LIN {X 0,Y 525.417,Z 230.64,A -85,B 0,C 180,E1 -4783.488,E2 -4783.488} C_VEL
LIN {X 0,Y 525.578,Z 217.368,A -85,B 0,C 180,E1 -4783.73,E2 -4783.73} C_VEL
LIN {X 0,Y 525.769,Z 127.353,A -85,B 0,C 180,E1 -4784.968,E2 -4784.968} C_VEL
LIN {X 0,Y 524.225,Z 116.388,A -85,B 0,C 180,E1 -4785.187,E2 -4785.187} C_VEL
LIN {X 0,Y 524.577,Z 97.639,A -85,B 0,C 180,E1 -4787.969,E2 -4787.969} C_VEL
LIN {X 0,Y 525.034,Z 77.543,A -85,B 0,C 180,E1 -4790.981,E2 -4790.981} C_VEL
LIN {X 0,Y 525.375,Z 61.269,A -85,B 0,C 180,E1 -4793.451,E2 -4793.451} C_VEL
LIN {X 0,Y 525.033,Z 57.51,A -85,B 0,C 180,E1 -4794.042,E2 -4794.042} C_VEL
LIN {X 0,Y 523.985,Z 52.216,A -85,B 0,C 180,E1 -4794.939,E2 -4794.939} C_VEL
LIN {X 0,Y 523.971,Z 52.218,A -85,B 0,C 180,E1 -4797.999,E2 -4797.999} C_VEL
LIN {X 0,Y 523.946,Z 52.215,A -85,B 0,C 180,E1 -4800.854,E2 -4800.854} C_VEL
LIN {X 0,Y 523.96,Z 52.22,A -85,B 0,C 180,E1 -4803.734,E2 -4803.734} C_VEL
LIN {X 0,Y 523.904,Z 52.222,A -85,B 0,C 180,E1 -4806.401,E2 -4806.401} C_VEL
LIN {X 0,Y 523.923,Z 52.219,A -85,B 0,C 180,E1 -4809.084,E2 -4809.084} C_VEL
LIN {X 0,Y 523.951,Z 52.217,A -85,B 0,C 180,E1 -4812.119,E2 -4812.119} C_VEL
LIN {X 0,Y 523.942,Z 52.222,A -85,B 0,C 180,E1 -4815.31,E2 -4815.31} C_VEL
LIN {X 0,Y 523.955,Z 52.215,A -85,B 0,C 180,E1 -4818.69,E2 -4818.69} C_VEL
LIN {X 0,Y 523.916,Z 52.224,A -85,B 0,C 180,E1 -4821.081,E2 -4821.081} C_VEL
LIN {X 0,Y 523.902,Z 52.222,A -85,B 0,C 180,E1 -4823.825,E2 -4823.825} C_VEL
LIN {X 0,Y 523.941,Z 52.218,A -85,B 0,C 180,E1 -4826.636,E2 -4826.636} C_VEL
LIN {X 0,Y 523.956,Z 52.218,A -85,B 0,C 180,E1 -4829.356,E2 -4829.356} C_VEL
LIN {X 0,Y 523.976,Z 52.212,A -85,B 0,C 180,E1 -4832.281,E2 -4832.281} C_VEL
LIN {X 0,Y 523.947,Z 52.219,A -85,B 0,C 180,E1 -4834.581,E2 -4834.581} C_VEL
LIN {X 0,Y 523.918,Z 52.218,A -85,B 0,C 180,E1 -4837.757,E2 -4837.757} C_VEL
LIN {X 0,Y 523.974,Z 52.216,A -85,B 0,C 180,E1 -4840.408,E2 -4840.408} C_VEL
LIN {X 0,Y 523.953,Z 52.22,A -85,B 0,C 180,E1 -4842.837,E2 -4842.837} C_VEL
LIN {X 0,Y 523.975,Z 52.212,A -85,B 0,C 180,E1 -4845.236,E2 -4845.236} C_VEL
LIN {X 0,Y 524.013,Z 52.215,A -85,B 0,C 180,E1 -4848.394,E2 -4848.394} C_VEL
LIN {X 0,Y 523.999,Z 52.209,A -85,B 0,C 180,E1 -4851.516,E2 -4851.516} C_VEL
LIN {X 0,Y 524.078,Z 52.202,A -85,B 0,C 180,E1 -4854.614,E2 -4854.614} C_VEL
LIN {X 0,Y 524.111,Z 52.197,A -85,B 0,C 180,E1 -4857.695,E2 -4857.695} C_VEL
LIN {X 0,Y 524.119,Z 52.194,A -85,B 0,C 180,E1 -4860.768,E2 -4860.768} C_VEL
LIN {X 0,Y 524.042,Z 52.203,A -85,B 0,C 180,E1 -4863.075,E2 -4863.075} C_VEL
LIN {X 0,Y 524.027,Z 52.21,A -85,B 0,C 180,E1 -4866.159,E2 -4866.159} C_VEL
LIN {X 0,Y 523.986,Z 52.212,A -85,B 0,C 180,E1 -4869.262,E2 -4869.262} C_VEL
LIN {X 0,Y 524,Z 52.217,A -85,B 0,C 180,E1 -4871.738,E2 -4871.738} C_VEL
LIN {X 0,Y 523.992,Z 52.211,A -85,B 0,C 180,E1 -4875.052,E2 -4875.052} C_VEL
LIN {X 0,Y 523.945,Z 52.218,A -85,B 0,C 180,E1 -4877.97,E2 -4877.97} C_VEL
LIN {X 0,Y 523.958,Z 52.213,A -85,B 0,C 180,E1 -4880.411,E2 -4880.411} C_VEL
LIN {X 0,Y 523.908,Z 52.222,A -85,B 0,C 180,E1 -4882.894,E2 -4882.894} C_VEL
LIN {X 0,Y 523.914,Z 52.226,A -85,B 0,C 180,E1 -4885.421,E2 -4885.421} C_VEL
LIN {X 0,Y 523.958,Z 52.214,A -85,B 0,C 180,E1 -4888,E2 -4888} C_VEL
LIN {X 0,Y 523.939,Z 52.221,A -85,B 0,C 180,E1 -4890.854,E2 -4890.854} C_VEL
LIN {X 0,Y 523.93,Z 52.218,A -85,B 0,C 180,E1 -4893.73,E2 -4893.73} C_VEL
LIN {X 0,Y 523.904,Z 52.222,A -85,B 0,C 180,E1 -4896.402,E2 -4896.402} C_VEL
LIN {X 0,Y 523.914,Z 52.225,A -85,B 0,C 180,E1 -4899.086,E2 -4899.086} C_VEL
LIN {X 0,Y 523.91,Z 52.221,A -85,B 0,C 180,E1 -4902.124,E2 -4902.124} C_VEL
LIN {X 0,Y 523.942,Z 52.217,A -85,B 0,C 180,E1 -4905.311,E2 -4905.311} C_VEL
LIN {X 0,Y 523.902,Z 52.225,A -85,B 0,C 180,E1 -4906.885,E2 -4906.885} C_VEL
LIN {X 0,Y 523.23,Z 52.307,A -85,B 0,C 180,E1 -4907.527,E2 -4907.527} C_VEL
LIN {X 0,Y 520.367,Z 52.67,A -85,B 0,C 180,E1 -4908.568,E2 -4908.568} C_VEL
LIN {X 0,Y 517.961,Z 52.965,A -85,B 0,C 180,E1 -4909.407,E2 -4909.407} C_VEL
LIN {X 0,Y 516.947,Z 53.09,A -85,B 0,C 180,E1 -4910.055,E2 -4910.055} C_VEL
LIN {X 0,Y 516.875,Z 53.101,A -85,B 0,C 180,E1 -4910.274,E2 -4910.274} C_VEL
LIN {X 0,Y 516.85,Z 53.099,A -85,B 0,C 180,E1 -4913.348,E2 -4913.348} C_VEL
LIN {X 0,Y 516.902,Z 53.098,A -85,B 0,C 180,E1 -4916.12,E2 -4916.12} C_VEL
LIN {X 0,Y 516.895,Z 53.094,A -85,B 0,C 180,E1 -4918.936,E2 -4918.936} C_VEL
LIN {X 0,Y 516.863,Z 53.099,A -85,B 0,C 180,E1 -4921.582,E2 -4921.582} C_VEL
LIN {X 0,Y 516.872,Z 53.103,A -85,B 0,C 180,E1 -4924.208,E2 -4924.208} C_VEL
LIN {X 0,Y 516.862,Z 53.098,A -85,B 0,C 180,E1 -4926.776,E2 -4926.776} C_VEL
LIN {X 0,Y 516.942,Z 53.094,A -85,B 0,C 180,E1 -4929.733,E2 -4929.733} C_VEL
LIN {X 0,Y 516.889,Z 53.095,A -85,B 0,C 180,E1 -4932.595,E2 -4932.595} C_VEL
LIN {X 0,Y 516.944,Z 53.091,A -85,B 0,C 180,E1 -4935.03,E2 -4935.03} C_VEL
LIN {X 0,Y 516.966,Z 53.271,A -85,B 0,C 180,E1 -4937.756,E2 -4937.756} C_VEL
LIN {X 0,Y 517.485,Z 57.551,A -85,B 0,C 180,E1 -4938.643,E2 -4938.643} C_VEL
LIN {X 0,Y 517.416,Z 69.345,A -85,B 0,C 180,E1 -4941.014,E2 -4941.014} C_VEL
LIN {X 0,Y 517.278,Z 72.801,A -85,B 0,C 180,E1 -4941.696,E2 -4941.696} C_VEL
LIN {X 0,Y 519.153,Z 83.02,A -85,B 0,C 180,E1 -4941.901,E2 -4941.901} C_VEL
LIN {X 0,Y 518.614,Z 179.674,A -85,B 0,C 180,E1 -4943.264,E2 -4943.264} C_VEL
LIN {X 0,Y 518.437,Z 193.363,A -85,B 0,C 180,E1 -4943.628,E2 -4943.628} C_VEL
LIN {X 0,Y 518.283,Z 205.634,A -85,B 0,C 180,E1 -4944.114,E2 -4944.114} C_VEL
LIN {X 0,Y 518.082,Z 217.393,A -85,B 0,C 180,E1 -4944.746,E2 -4944.746} C_VEL
LIN {X 0,Y 517.745,Z 228.688,A -85,B 0,C 180,E1 -4945.524,E2 -4945.524} C_VEL
LIN {X 0,Y 517.419,Z 238.884,A -85,B 0,C 180,E1 -4946.399,E2 -4946.399} C_VEL
LIN {X 0,Y 517.184,Z 247.231,A -85,B 0,C 180,E1 -4947.274,E2 -4947.274} C_VEL
LIN {X 0,Y 516.859,Z 256.313,A -85,B 0,C 180,E1 -4948.442,E2 -4948.442} C_VEL
LIN {X 0,Y 516.712,Z 263.613,A -85,B 0,C 180,E1 -4949.611,E2 -4949.611} C_VEL
LIN {X 0,Y 516.473,Z 269.502,A -85,B 0,C 180,E1 -4950.78,E2 -4950.78} C_VEL
LIN {X 0,Y 516.401,Z 274.157,A -85,B 0,C 180,E1 -4951.95,E2 -4951.95} C_VEL
LIN {X 0,Y 516.389,Z 277.725,A -85,B 0,C 180,E1 -4953.121,E2 -4953.121} C_VEL
LIN {X 0,Y 516.332,Z 279.576,A -85,B 0,C 180,E1 -4953.903,E2 -4953.903} C_VEL
LIN {X 0,Y 516.247,Z 280.97,A -85,B 0,C 180,E1 -4954.685,E2 -4954.685} C_VEL
LIN {X 0,Y 516.312,Z 281.956,A -85,B 0,C 180,E1 -4955.468,E2 -4955.468} C_VEL
LIN {X 0,Y 516.374,Z 282.679,A -85,B 0,C 180,E1 -4956.506,E2 -4956.506} C_VEL
LIN {X 0,Y 516.279,Z 282.577,A -85,B 0,C 180,E1 -4957.824,E2 -4957.824} C_VEL
LIN {X 0,Y 516.23,Z 280.982,A -85,B 0,C 180,E1 -4959.403,E2 -4959.403} C_VEL
LIN {X 0,Y 516.294,Z 279.577,A -85,B 0,C 180,E1 -4960.193,E2 -4960.193} C_VEL
LIN {X 0,Y 516.366,Z 276.299,A -85,B 0,C 180,E1 -4961.488,E2 -4961.488} C_VEL
LIN {X 0,Y 516.474,Z 272.599,A -85,B 0,C 180,E1 -4962.576,E2 -4962.576} C_VEL
LIN {X 0,Y 516.644,Z 266.35,A -85,B 0,C 180,E1 -4963.973,E2 -4963.973} C_VEL
LIN {X 0,Y 516.797,Z 260.069,A -85,B 0,C 180,E1 -4965.083,E2 -4965.083} C_VEL
LIN {X 0,Y 517.008,Z 252.455,A -85,B 0,C 180,E1 -4966.181,E2 -4966.181} C_VEL
LIN {X 0,Y 517.251,Z 243.92,A -85,B 0,C 180,E1 -4967.189,E2 -4967.189} C_VEL
LIN {X 0,Y 517.561,Z 233.283,A -85,B 0,C 180,E1 -4968.199,E2 -4968.199} C_VEL
LIN {X 0,Y 517.868,Z 222.67,A -85,B 0,C 180,E1 -4969.009,E2 -4969.009} C_VEL
LIN {X 0,Y 518.182,Z 210.921,A -85,B 0,C 180,E1 -4969.717,E2 -4969.717} C_VEL
LIN {X 0,Y 518.418,Z 198.575,A -85,B 0,C 180,E1 -4970.276,E2 -4970.276} C_VEL
LIN {X 0,Y 518.614,Z 186.111,A -85,B 0,C 180,E1 -4970.678,E2 -4970.678} C_VEL
LIN {X 0,Y 518.725,Z 174.043,A -85,B 0,C 180,E1 -4970.924,E2 -4970.924} C_VEL
LIN {X 0,Y 519.058,Z 81.453,A -85,B 0,C 180,E1 -4972.218,E2 -4972.218} C_VEL
LIN {X 0,Y 517.329,Z 72.818,A -85,B 0,C 180,E1 -4972.41,E2 -4972.41} C_VEL
LIN {X 0,Y 517.6,Z 58.332,A -85,B 0,C 180,E1 -4975.323,E2 -4975.323} C_VEL
LIN {X 0,Y 516.886,Z 53.103,A -85,B 0,C 180,E1 -4976.462,E2 -4976.462} C_VEL
LIN {X 0,Y 516.889,Z 53.098,A -85,B 0,C 180,E1 -4979.518,E2 -4979.518} C_VEL
LIN {X 0,Y 516.868,Z 53.104,A -85,B 0,C 180,E1 -4982.538,E2 -4982.538} C_VEL
LIN {X 0,Y 516.831,Z 53.103,A -85,B 0,C 180,E1 -4985.323,E2 -4985.323} C_VEL
LIN {X 0,Y 516.862,Z 53.1,A -85,B 0,C 180,E1 -4988.718,E2 -4988.718} C_VEL
LIN {X 0,Y 516.834,Z 53.109,A -85,B 0,C 180,E1 -4991.783,E2 -4991.783} C_VEL
LIN {X 0,Y 516.9,Z 53.089,A -85,B 0,C 180,E1 -4995.007,E2 -4995.007} C_VEL
LIN {X 0,Y 516.832,Z 53.101,A -85,B 0,C 180,E1 -4998.409,E2 -4998.409} C_VEL
LIN {X 0,Y 516.849,Z 53.104,A -85,B 0,C 180,E1 -5001.281,E2 -5001.281} C_VEL
LIN {X 0,Y 516.83,Z 53.101,A -85,B 0,C 180,E1 -5004.677,E2 -5004.677} C_VEL
LIN {X 0,Y 516.867,Z 53.102,A -85,B 0,C 180,E1 -5007.462,E2 -5007.462} C_VEL
LIN {X 0,Y 516.848,Z 53.1,A -85,B 0,C 180,E1 -5010.489,E2 -5010.489} C_VEL
LIN {X 0,Y 516.829,Z 53.108,A -85,B 0,C 180,E1 -5013.337,E2 -5013.337} C_VEL
LIN {X 0,Y 516.871,Z 53.096,A -85,B 0,C 180,E1 -5015.926,E2 -5015.926} C_VEL
LIN {X 0,Y 516.886,Z 53.095,A -85,B 0,C 180,E1 -5018.462,E2 -5018.462} C_VEL
LIN {X 0,Y 516.888,Z 53.1,A -85,B 0,C 180,E1 -5020.954,E2 -5020.954} C_VEL
LIN {X 0,Y 516.882,Z 53.096,A -85,B 0,C 180,E1 -5023.409,E2 -5023.409} C_VEL
LIN {X 0,Y 516.872,Z 53.097,A -85,B 0,C 180,E1 -5025.833,E2 -5025.833} C_VEL
LIN {X 0,Y 516.946,Z 53.089,A -85,B 0,C 180,E1 -5029.028,E2 -5029.028} C_VEL
LIN {X 0,Y 516.93,Z 53.094,A -85,B 0,C 180,E1 -5032.186,E2 -5032.186} C_VEL
LIN {X 0,Y 516.983,Z 53.088,A -85,B 0,C 180,E1 -5034.539,E2 -5034.539} C_VEL
LIN {X 0,Y 517.077,Z 53.073,A -85,B 0,C 180,E1 -5037.663,E2 -5037.663} C_VEL
LIN {X 0,Y 517.092,Z 53.069,A -85,B 0,C 180,E1 -5040.779,E2 -5040.779} C_VEL
LIN {X 0,Y 516.949,Z 53.087,A -85,B 0,C 180,E1 -5043.117,E2 -5043.117} C_VEL
LIN {X 0,Y 516.976,Z 53.086,A -85,B 0,C 180,E1 -5046.243,E2 -5046.243} C_VEL
LIN {X 0,Y 516.941,Z 53.091,A -85,B 0,C 180,E1 -5049.389,E2 -5049.389} C_VEL
LIN {X 0,Y 516.956,Z 53.09,A -85,B 0,C 180,E1 -5051.807,E2 -5051.807} C_VEL
LIN {X 0,Y 516.942,Z 53.09,A -85,B 0,C 180,E1 -5055.144,E2 -5055.144} C_VEL
LIN {X 0,Y 516.881,Z 53.095,A -85,B 0,C 180,E1 -5058.224,E2 -5058.224} C_VEL
LIN {X 0,Y 516.908,Z 53.092,A -85,B 0,C 180,E1 -5060.702,E2 -5060.702} C_VEL
LIN {X 0,Y 516.888,Z 53.095,A -85,B 0,C 180,E1 -5064.073,E2 -5064.073} C_VEL
LIN {X 0,Y 516.907,Z 53.093,A -85,B 0,C 180,E1 -5066.659,E2 -5066.659} C_VEL
LIN {X 0,Y 516.91,Z 53.095,A -85,B 0,C 180,E1 -5069.523,E2 -5069.523} C_VEL
LIN {X 0,Y 516.899,Z 53.095,A -85,B 0,C 180,E1 -5072.543,E2 -5072.543} C_VEL
LIN {X 0,Y 516.871,Z 53.094,A -85,B 0,C 180,E1 -5075.33,E2 -5075.33} C_VEL
LIN {X 0,Y 516.882,Z 53.093,A -85,B 0,C 180,E1 -5077.943,E2 -5077.943} C_VEL
LIN {X 0,Y 516.886,Z 53.102,A -85,B 0,C 180,E1 -5080.742,E2 -5080.742} C_VEL
LIN {X 0,Y 516.885,Z 53.102,A -85,B 0,C 180,E1 -5082.831,E2 -5082.831} C_VEL
LIN {X 0,Y 516.898,Z 53.096,A -85,B 0,C 180,E1 -5085.007,E2 -5085.007} C_VEL
LIN {X 0,Y 516.916,Z 53.097,A -85,B 0,C 180,E1 -5088.399,E2 -5088.399} C_VEL
LIN {X 0,Y 516.884,Z 53.095,A -85,B 0,C 180,E1 -5091.284,E2 -5091.284} C_VEL
LIN {X 0,Y 516.874,Z 53.102,A -85,B 0,C 180,E1 -5094.22,E2 -5094.22} C_VEL
LIN {X 0,Y 516.898,Z 53.097,A -85,B 0,C 180,E1 -5097.053,E2 -5097.053} C_VEL
LIN {X 0,Y 516.895,Z 53.102,A -85,B 0,C 180,E1 -5099.796,E2 -5099.796} C_VEL
LIN {X 0,Y 516.929,Z 53.094,A -85,B 0,C 180,E1 -5102.467,E2 -5102.467} C_VEL
LIN {X 0,Y 516.939,Z 53.134,A -85,B 0,C 180,E1 -5104.858,E2 -5104.858} C_VEL
LIN {X 0,Y 518.443,Z 61.217,A -85,B 0,C 180,E1 -5106.216,E2 -5106.216} C_VEL
LIN {X 0,Y 518.131,Z 74.628,A -85,B 0,C 180,E1 -5108.307,E2 -5108.307} C_VEL
LIN {X 0,Y 517.731,Z 90.731,A -85,B 0,C 180,E1 -5110.78,E2 -5110.78} C_VEL
LIN {X 0,Y 517.337,Z 109.522,A -85,B 0,C 180,E1 -5113.627,E2 -5113.627} C_VEL
LIN {X 0,Y 517.18,Z 116.074,A -85,B 0,C 180,E1 -5114.61,E2 -5114.61} C_VEL
LIN {X 0,Y 519.009,Z 129.152,A -85,B 0,C 180,E1 -5114.863,E2 -5114.863} C_VEL
LIN {X 0,Y 518.575,Z 224.633,A -85,B 0,C 180,E1 -5116.205,E2 -5116.205} C_VEL
LIN {X 0,Y 518.337,Z 237.966,A -85,B 0,C 180,E1 -5116.549,E2 -5116.549} C_VEL
LIN {X 0,Y 518.029,Z 251.299,A -85,B 0,C 180,E1 -5117.064,E2 -5117.064} C_VEL
LIN {X 0,Y 517.755,Z 263.311,A -85,B 0,C 180,E1 -5117.706,E2 -5117.706} C_VEL
LIN {X 0,Y 517.445,Z 274.128,A -85,B 0,C 180,E1 -5118.443,E2 -5118.443} C_VEL
LIN {X 0,Y 517.173,Z 284.608,A -85,B 0,C 180,E1 -5119.33,E2 -5119.33} C_VEL
LIN {X 0,Y 516.878,Z 293.178,A -85,B 0,C 180,E1 -5120.214,E2 -5120.214} C_VEL
LIN {X 0,Y 516.672,Z 301.089,A -85,B 0,C 180,E1 -5121.197,E2 -5121.197} C_VEL
LIN {X 0,Y 516.511,Z 308.82,A -85,B 0,C 180,E1 -5122.376,E2 -5122.376} C_VEL
LIN {X 0,Y 516.353,Z 315.946,A -85,B 0,C 180,E1 -5123.749,E2 -5123.749} C_VEL
LIN {X 0,Y 516.311,Z 320.69,A -85,B 0,C 180,E1 -5124.924,E2 -5124.924} C_VEL
LIN {X 0,Y 516.351,Z 324.319,A -85,B 0,C 180,E1 -5126.098,E2 -5126.098} C_VEL
LIN {X 0,Y 516.303,Z 326.188,A -85,B 0,C 180,E1 -5126.879,E2 -5126.879} C_VEL
LIN {X 0,Y 516.264,Z 327.59,A -85,B 0,C 180,E1 -5127.659,E2 -5127.659} C_VEL
LIN {X 0,Y 516.177,Z 329.2,A -85,B 0,C 180,E1 -5129.22,E2 -5129.22} C_VEL
LIN {X 0,Y 516.179,Z 329.419,A -85,B 0,C 180,E1 -5130,E2 -5130} C_VEL
LIN {X 0,Y 516.196,Z 328.597,A -85,B 0,C 180,E1 -5131.56,E2 -5131.56} C_VEL
LIN {X 0,Y 516.264,Z 327.603,A -85,B 0,C 180,E1 -5132.34,E2 -5132.34} C_VEL
LIN {X 0,Y 516.303,Z 326.205,A -85,B 0,C 180,E1 -5133.121,E2 -5133.121} C_VEL
LIN {X 0,Y 516.309,Z 323.26,A -85,B 0,C 180,E1 -5134.293,E2 -5134.293} C_VEL
LIN {X 0,Y 516.364,Z 319.275,A -85,B 0,C 180,E1 -5135.467,E2 -5135.467} C_VEL
LIN {X 0,Y 516.414,Z 313.144,A -85,B 0,C 180,E1 -5136.839,E2 -5136.839} C_VEL
LIN {X 0,Y 516.561,Z 306.446,A -85,B 0,C 180,E1 -5138.016,E2 -5138.016} C_VEL
LIN {X 0,Y 516.741,Z 298.137,A -85,B 0,C 180,E1 -5139.195,E2 -5139.195} C_VEL
LIN {X 0,Y 516.947,Z 289.622,A -85,B 0,C 180,E1 -5140.18,E2 -5140.18} C_VEL
LIN {X 0,Y 517.29,Z 279.107,A -85,B 0,C 180,E1 -5141.163,E2 -5141.163} C_VEL
LIN {X 0,Y 517.607,Z 267.374,A -85,B 0,C 180,E1 -5142.043,E2 -5142.043} C_VEL
LIN {X 0,Y 517.946,Z 255.379,A -85,B 0,C 180,E1 -5142.738,E2 -5142.738} C_VEL
LIN {X 0,Y 518.209,Z 243.005,A -85,B 0,C 180,E1 -5143.28,E2 -5143.28} C_VEL
LIN {X 0,Y 518.53,Z 230.312,A -85,B 0,C 180,E1 -5143.671,E2 -5143.671} C_VEL
LIN {X 0,Y 518.677,Z 217.028,A -85,B 0,C 180,E1 -5143.916,E2 -5143.916} C_VEL
LIN {X 0,Y 518.96,Z 128.491,A -85,B 0,C 180,E1 -5145.149,E2 -5145.149} C_VEL
LIN {X 0,Y 517.219,Z 116.148,A -85,B 0,C 180,E1 -5145.387,E2 -5145.387} C_VEL
LIN {X 0,Y 517.662,Z 96.105,A -85,B 0,C 180,E1 -5148.4,E2 -5148.4} C_VEL
LIN {X 0,Y 518.122,Z 75.816,A -85,B 0,C 180,E1 -5151.484,E2 -5151.484} C_VEL
LIN {X 0,Y 518.441,Z 62.24,A -85,B 0,C 180,E1 -5153.572,E2 -5153.572} C_VEL
LIN {X 0,Y 517.434,Z 55.557,A -85,B 0,C 180,E1 -5154.656,E2 -5154.656} C_VEL
LIN {X 0,Y 516.948,Z 53.092,A -85,B 0,C 180,E1 -5155.087,E2 -5155.087} C_VEL
LIN {X 0,Y 516.928,Z 53.094,A -85,B 0,C 180,E1 -5157.905,E2 -5157.905} C_VEL
LIN {X 0,Y 516.893,Z 53.1,A -85,B 0,C 180,E1 -5160.203,E2 -5160.203} C_VEL
LIN {X 0,Y 516.896,Z 53.093,A -85,B 0,C 180,E1 -5162.947,E2 -5162.947} C_VEL
LIN {X 0,Y 516.872,Z 53.105,A -85,B 0,C 180,E1 -5165.78,E2 -5165.78} C_VEL
LIN {X 0,Y 516.883,Z 53.095,A -85,B 0,C 180,E1 -5168.715,E2 -5168.715} C_VEL
LIN {X 0,Y 516.912,Z 53.098,A -85,B 0,C 180,E1 -5171.775,E2 -5171.775} C_VEL
LIN {X 0,Y 516.895,Z 53.096,A -85,B 0,C 180,E1 -5175.007,E2 -5175.007} C_VEL
LIN {X 0,Y 516.913,Z 53.091,A -85,B 0,C 180,E1 -5178.399,E2 -5178.399} C_VEL
LIN {X 0,Y 516.879,Z 53.104,A -85,B 0,C 180,E1 -5181.284,E2 -5181.284} C_VEL
LIN {X 0,Y 516.873,Z 53.096,A -85,B 0,C 180,E1 -5184.22,E2 -5184.22} C_VEL
LIN {X 0,Y 516.895,Z 53.101,A -85,B 0,C 180,E1 -5187.053,E2 -5187.053} C_VEL
LIN {X 0,Y 516.891,Z 53.094,A -85,B 0,C 180,E1 -5189.796,E2 -5189.796} C_VEL
LIN {X 0,Y 516.926,Z 53.092,A -85,B 0,C 180,E1 -5192.467,E2 -5192.467} C_VEL
LIN {X 0,Y 516.903,Z 53.098,A -85,B 0,C 180,E1 -5195.072,E2 -5195.072} C_VEL
LIN {X 0,Y 516.885,Z 53.099,A -85,B 0,C 180,E1 -5198.462,E2 -5198.462} C_VEL
LIN {X 0,Y 516.9,Z 53.098,A -85,B 0,C 180,E1 -5200.955,E2 -5200.955} C_VEL
LIN {X 0,Y 516.903,Z 53.093,A -85,B 0,C 180,E1 -5203.41,E2 -5203.41} C_VEL
LIN {X 0,Y 516.891,Z 53.095,A -85,B 0,C 180,E1 -5205.834,E2 -5205.834} C_VEL
LIN {X 0,Y 516.95,Z 53.088,A -85,B 0,C 180,E1 -5209.028,E2 -5209.028} C_VEL
LIN {X 0,Y 516.977,Z 53.09,A -85,B 0,C 180,E1 -5212.187,E2 -5212.187} C_VEL
LIN {X 0,Y 517.026,Z 53.082,A -85,B 0,C 180,E1 -5214.54,E2 -5214.54} C_VEL
LIN {X 0,Y 517.082,Z 53.072,A -85,B 0,C 180,E1 -5217.663,E2 -5217.663} C_VEL
LIN {X 0,Y 517.09,Z 53.07,A -85,B 0,C 180,E1 -5220.779,E2 -5220.779} C_VEL
LIN {X 0,Y 516.985,Z 53.082,A -85,B 0,C 180,E1 -5223.117,E2 -5223.117} C_VEL
LIN {X 0,Y 516.989,Z 53.086,A -85,B 0,C 180,E1 -5226.244,E2 -5226.244} C_VEL
LIN {X 0,Y 516.942,Z 53.091,A -85,B 0,C 180,E1 -5229.39,E2 -5229.39} C_VEL
LIN {X 0,Y 516.952,Z 53.094,A -85,B 0,C 180,E1 -5231.807,E2 -5231.807} C_VEL
LIN {X 0,Y 516.943,Z 53.09,A -85,B 0,C 180,E1 -5235.146,E2 -5235.146} C_VEL
LIN {X 0,Y 516.913,Z 53.092,A -85,B 0,C 180,E1 -5238.223,E2 -5238.223} C_VEL
LIN {X 0,Y 516.905,Z 53.093,A -85,B 0,C 180,E1 -5240.702,E2 -5240.702} C_VEL
LIN {X 0,Y 516.886,Z 53.095,A -85,B 0,C 180,E1 -5244.074,E2 -5244.074} C_VEL
LIN {X 0,Y 516.908,Z 53.093,A -85,B 0,C 180,E1 -5246.659,E2 -5246.659} C_VEL
LIN {X 0,Y 516.909,Z 53.095,A -85,B 0,C 180,E1 -5249.524,E2 -5249.524} C_VEL
LIN {X 0,Y 516.895,Z 53.096,A -85,B 0,C 180,E1 -5252.543,E2 -5252.543} C_VEL
LIN {X 0,Y 516.866,Z 53.101,A -85,B 0,C 180,E1 -5255.33,E2 -5255.33} C_VEL
LIN {X 0,Y 516.88,Z 53.095,A -85,B 0,C 180,E1 -5257.943,E2 -5257.943} C_VEL
LIN {X 0,Y 516.854,Z 53.107,A -85,B 0,C 180,E1 -5260.745,E2 -5260.745} C_VEL
LIN {X 0,Y 516.882,Z 53.095,A -85,B 0,C 180,E1 -5263.904,E2 -5263.904} C_VEL
LIN {X 0,Y 516.849,Z 53.099,A -85,B 0,C 180,E1 -5266.887,E2 -5266.887} C_VEL
LIN {X 0,Y 516.882,Z 53.095,A -85,B 0,C 180,E1 -5269.591,E2 -5269.591} C_VEL
LIN {X 0,Y 516.875,Z 53.101,A -85,B 0,C 180,E1 -5270.274,E2 -5270.274} C_VEL
LIN {X 0,Y 516.232,Z 53.187,A -85,B 0,C 180,E1 -5270.925,E2 -5270.925} C_VEL
LIN {X 0,Y 513.378,Z 53.54,A -85,B 0,C 180,E1 -5271.98,E2 -5271.98} C_VEL
LIN {X 0,Y 510.944,Z 53.838,A -85,B 0,C 180,E1 -5272.83,E2 -5272.83} C_VEL
LIN {X 0,Y 509.892,Z 53.966,A -85,B 0,C 180,E1 -5273.487,E2 -5273.487} C_VEL
LIN {X 0,Y 509.804,Z 53.977,A -85,B 0,C 180,E1 -5273.709,E2 -5273.709} C_VEL
LIN {X 0,Y 509.855,Z 53.976,A -85,B 0,C 180,E1 -5276.539,E2 -5276.539} C_VEL
LIN {X 0,Y 509.849,Z 53.971,A -85,B 0,C 180,E1 -5279.335,E2 -5279.335} C_VEL
LIN {X 0,Y 509.847,Z 53.979,A -85,B 0,C 180,E1 -5282.052,E2 -5282.052} C_VEL
LIN {X 0,Y 509.804,Z 53.978,A -85,B 0,C 180,E1 -5284.7,E2 -5284.7} C_VEL
LIN {X 0,Y 509.83,Z 53.976,A -85,B 0,C 180,E1 -5287.459,E2 -5287.459} C_VEL
LIN {X 0,Y 509.919,Z 53.971,A -85,B 0,C 180,E1 -5289.845,E2 -5289.845} C_VEL
LIN {X 0,Y 509.86,Z 53.971,A -85,B 0,C 180,E1 -5293.174,E2 -5293.174} C_VEL
LIN {X 0,Y 509.858,Z 53.979,A -85,B 0,C 180,E1 -5295.634,E2 -5295.634} C_VEL
LIN {X 0,Y 509.908,Z 54.059,A -85,B 0,C 180,E1 -5297.615,E2 -5297.615} C_VEL
LIN {X 0,Y 510.464,Z 58.208,A -85,B 0,C 180,E1 -5298.485,E2 -5298.485} C_VEL
LIN {X 0,Y 510.427,Z 70.066,A -85,B 0,C 180,E1 -5300.89,E2 -5300.89} C_VEL
LIN {X 0,Y 510.297,Z 73.056,A -85,B 0,C 180,E1 -5301.484,E2 -5301.484} C_VEL
LIN {X 0,Y 512.301,Z 83.987,A -85,B 0,C 180,E1 -5301.709,E2 -5301.709} C_VEL
LIN {X 0,Y 511.733,Z 179.747,A -85,B 0,C 180,E1 -5303.074,E2 -5303.074} C_VEL
LIN {X 0,Y 511.565,Z 192.771,A -85,B 0,C 180,E1 -5303.418,E2 -5303.418} C_VEL
LIN {X 0,Y 511.376,Z 205.848,A -85,B 0,C 180,E1 -5303.936,E2 -5303.936} C_VEL
LIN {X 0,Y 511.153,Z 217.649,A -85,B 0,C 180,E1 -5304.576,E2 -5304.576} C_VEL
LIN {X 0,Y 510.799,Z 228.966,A -85,B 0,C 180,E1 -5305.364,E2 -5305.364} C_VEL
LIN {X 0,Y 510.453,Z 239.172,A -85,B 0,C 180,E1 -5306.25,E2 -5306.25} C_VEL
LIN {X 0,Y 510.155,Z 248.374,A -85,B 0,C 180,E1 -5307.237,E2 -5307.237} C_VEL
LIN {X 0,Y 509.814,Z 257.287,A -85,B 0,C 180,E1 -5308.42,E2 -5308.42} C_VEL
LIN {X 0,Y 509.668,Z 264.473,A -85,B 0,C 180,E1 -5309.605,E2 -5309.605} C_VEL
LIN {X 0,Y 509.397,Z 270.263,A -85,B 0,C 180,E1 -5310.791,E2 -5310.791} C_VEL
LIN {X 0,Y 509.336,Z 274.823,A -85,B 0,C 180,E1 -5311.977,E2 -5311.977} C_VEL
LIN {X 0,Y 509.325,Z 278.304,A -85,B 0,C 180,E1 -5313.164,E2 -5313.164} C_VEL
LIN {X 0,Y 509.258,Z 280.083,A -85,B 0,C 180,E1 -5313.957,E2 -5313.957} C_VEL
LIN {X 0,Y 509.162,Z 281.428,A -85,B 0,C 180,E1 -5314.751,E2 -5314.751} C_VEL
LIN {X 0,Y 509.245,Z 282.373,A -85,B 0,C 180,E1 -5315.544,E2 -5315.544} C_VEL
LIN {X 0,Y 509.291,Z 282.998,A -85,B 0,C 180,E1 -5316.497,E2 -5316.497} C_VEL
LIN {X 0,Y 509.186,Z 282.839,A -85,B 0,C 180,E1 -5317.934,E2 -5317.934} C_VEL
LIN {X 0,Y 509.146,Z 281.164,A -85,B 0,C 180,E1 -5319.535,E2 -5319.535} C_VEL
LIN {X 0,Y 509.231,Z 279.679,A -85,B 0,C 180,E1 -5320.336,E2 -5320.336} C_VEL
LIN {X 0,Y 509.288,Z 276.651,A -85,B 0,C 180,E1 -5321.54,E2 -5321.54} C_VEL
LIN {X 0,Y 509.408,Z 272.523,A -85,B 0,C 180,E1 -5322.753,E2 -5322.753} C_VEL
LIN {X 0,Y 509.618,Z 266.168,A -85,B 0,C 180,E1 -5324.169,E2 -5324.169} C_VEL
LIN {X 0,Y 509.8,Z 259.201,A -85,B 0,C 180,E1 -5325.39,E2 -5325.39} C_VEL
LIN {X 0,Y 510.061,Z 250.393,A -85,B 0,C 180,E1 -5326.613,E2 -5326.613} C_VEL
LIN {X 0,Y 510.384,Z 241.305,A -85,B 0,C 180,E1 -5327.635,E2 -5327.635} C_VEL
LIN {X 0,Y 510.656,Z 231.244,A -85,B 0,C 180,E1 -5328.558,E2 -5328.558} C_VEL
LIN {X 0,Y 510.991,Z 219.985,A -85,B 0,C 180,E1 -5329.379,E2 -5329.379} C_VEL
LIN {X 0,Y 511.34,Z 207.269,A -85,B 0,C 180,E1 -5330.097,E2 -5330.097} C_VEL
LIN {X 0,Y 511.605,Z 194.929,A -85,B 0,C 180,E1 -5330.611,E2 -5330.611} C_VEL
LIN {X 0,Y 511.8,Z 182.356,A -85,B 0,C 180,E1 -5330.968,E2 -5330.968} C_VEL
LIN {X 0,Y 511.924,Z 162.179,A -85,B 0,C 180,E1 -5331.292,E2 -5331.292} C_VEL
LIN {X 0,Y 512.238,Z 82.329,A -85,B 0,C 180,E1 -5332.424,E2 -5332.424} C_VEL
LIN {X 0,Y 510.354,Z 73.134,A -85,B 0,C 180,E1 -5332.629,E2 -5332.629} C_VEL
LIN {X 0,Y 510.629,Z 59.14,A -85,B 0,C 180,E1 -5335.475,E2 -5335.475} C_VEL
LIN {X 0,Y 509.869,Z 53.978,A -85,B 0,C 180,E1 -5336.585,E2 -5336.585} C_VEL
LIN {X 0,Y 509.831,Z 53.978,A -85,B 0,C 180,E1 -5339.753,E2 -5339.753} C_VEL
LIN {X 0,Y 509.826,Z 53.979,A -85,B 0,C 180,E1 -5342.765,E2 -5342.765} C_VEL
LIN {X 0,Y 509.783,Z 53.983,A -85,B 0,C 180,E1 -5345.571,E2 -5345.571} C_VEL
LIN {X 0,Y 509.811,Z 53.982,A -85,B 0,C 180,E1 -5348.342,E2 -5348.342} C_VEL
LIN {X 0,Y 509.786,Z 53.983,A -85,B 0,C 180,E1 -5351.433,E2 -5351.433} C_VEL
LIN {X 0,Y 509.838,Z 53.968,A -85,B 0,C 180,E1 -5354.67,E2 -5354.67} C_VEL
LIN {X 0,Y 509.789,Z 53.986,A -85,B 0,C 180,E1 -5357.505,E2 -5357.505} C_VEL
LIN {X 0,Y 509.806,Z 53.977,A -85,B 0,C 180,E1 -5360.643,E2 -5360.643} C_VEL
LIN {X 0,Y 509.757,Z 53.988,A -85,B 0,C 180,E1 -5363.641,E2 -5363.641} C_VEL
LIN {X 0,Y 509.827,Z 53.975,A -85,B 0,C 180,E1 -5366.536,E2 -5366.536} C_VEL
LIN {X 0,Y 509.805,Z 53.984,A -85,B 0,C 180,E1 -5369.331,E2 -5369.331} C_VEL
LIN {X 0,Y 509.827,Z 53.973,A -85,B 0,C 180,E1 -5372.05,E2 -5372.05} C_VEL
LIN {X 0,Y 509.784,Z 53.983,A -85,B 0,C 180,E1 -5374.699,E2 -5374.699} C_VEL
LIN {X 0,Y 509.828,Z 53.975,A -85,B 0,C 180,E1 -5377.459,E2 -5377.459} C_VEL
LIN {X 0,Y 509.911,Z 53.964,A -85,B 0,C 180,E1 -5379.844,E2 -5379.844} C_VEL
LIN {X 0,Y 509.855,Z 53.973,A -85,B 0,C 180,E1 -5383.173,E2 -5383.173} C_VEL
LIN {X 0,Y 509.846,Z 53.972,A -85,B 0,C 180,E1 -5385.633,E2 -5385.633} C_VEL
LIN {X 0,Y 509.91,Z 53.967,A -85,B 0,C 180,E1 -5388.874,E2 -5388.874} C_VEL
LIN {X 0,Y 509.882,Z 53.971,A -85,B 0,C 180,E1 -5392.077,E2 -5392.077} C_VEL
LIN {X 0,Y 509.936,Z 53.965,A -85,B 0,C 180,E1 -5394.464,E2 -5394.464} C_VEL
LIN {X 0,Y 510.048,Z 53.948,A -85,B 0,C 180,E1 -5397.631,E2 -5397.631} C_VEL
LIN {X 0,Y 510.041,Z 53.947,A -85,B 0,C 180,E1 -5400.789,E2 -5400.789} C_VEL
LIN {X 0,Y 509.894,Z 53.966,A -85,B 0,C 180,E1 -5403.16,E2 -5403.16} C_VEL
LIN {X 0,Y 509.924,Z 53.963,A -85,B 0,C 180,E1 -5406.33,E2 -5406.33} C_VEL
LIN {X 0,Y 509.881,Z 53.971,A -85,B 0,C 180,E1 -5409.521,E2 -5409.521} C_VEL
LIN {X 0,Y 509.908,Z 53.967,A -85,B 0,C 180,E1 -5411.931,E2 -5411.931} C_VEL
LIN {X 0,Y 509.898,Z 53.968,A -85,B 0,C 180,E1 -5415.242,E2 -5415.242} C_VEL
LIN {X 0,Y 509.841,Z 53.971,A -85,B 0,C 180,E1 -5418.484,E2 -5418.484} C_VEL
LIN {X 0,Y 509.849,Z 53.974,A -85,B 0,C 180,E1 -5421.002,E2 -5421.002} C_VEL
LIN {X 0,Y 509.822,Z 53.981,A -85,B 0,C 180,E1 -5423.564,E2 -5423.564} C_VEL
LIN {X 0,Y 509.881,Z 53.966,A -85,B 0,C 180,E1 -5426.371,E2 -5426.371} C_VEL
LIN {X 0,Y 509.874,Z 53.973,A -85,B 0,C 180,E1 -5428.844,E2 -5428.844} C_VEL
LIN {X 0,Y 509.821,Z 53.977,A -85,B 0,C 180,E1 -5431.59,E2 -5431.59} C_VEL
LIN {X 0,Y 509.852,Z 53.973,A -85,B 0,C 180,E1 -5434.413,E2 -5434.413} C_VEL
LIN {X 0,Y 509.819,Z 53.975,A -85,B 0,C 180,E1 -5437.341,E2 -5437.341} C_VEL
LIN {X 0,Y 509.841,Z 53.977,A -85,B 0,C 180,E1 -5440.382,E2 -5440.382} C_VEL
LIN {X 0,Y 509.825,Z 53.978,A -85,B 0,C 180,E1 -5443.062,E2 -5443.062} C_VEL
LIN {X 0,Y 509.825,Z 53.975,A -85,B 0,C 180,E1 -5445.793,E2 -5445.793} C_VEL
LIN {X 0,Y 509.858,Z 53.977,A -85,B 0,C 180,E1 -5448.574,E2 -5448.574} C_VEL
LIN {X 0,Y 509.854,Z 53.973,A -85,B 0,C 180,E1 -5451.786,E2 -5451.786} C_VEL
LIN {X 0,Y 509.833,Z 53.978,A -85,B 0,C 180,E1 -5454.622,E2 -5454.622} C_VEL
LIN {X 0,Y 509.864,Z 53.974,A -85,B 0,C 180,E1 -5457.481,E2 -5457.481} C_VEL
LIN {X 0,Y 509.861,Z 53.979,A -85,B 0,C 180,E1 -5460.274,E2 -5460.274} C_VEL
LIN {X 0,Y 509.887,Z 53.97,A -85,B 0,C 180,E1 -5462.944,E2 -5462.944} C_VEL
LIN {X 0,Y 509.876,Z 53.974,A -85,B 0,C 180,E1 -5464.649,E2 -5464.649} C_VEL
LIN {X 0,Y 511.595,Z 63.719,A -85,B 0,C 180,E1 -5466.308,E2 -5466.308} C_VEL
LIN {X 0,Y 511.019,Z 83.203,A -85,B 0,C 180,E1 -5469.375,E2 -5469.375} C_VEL
LIN {X 0,Y 510.47,Z 103.892,A -85,B 0,C 180,E1 -5472.575,E2 -5472.575} C_VEL
LIN {X 0,Y 510.208,Z 115.965,A -85,B 0,C 180,E1 -5474.405,E2 -5474.405} C_VEL
LIN {X 0,Y 512.152,Z 130.25,A -85,B 0,C 180,E1 -5474.671,E2 -5474.671} C_VEL
LIN {X 0,Y 511.692,Z 224.405,A -85,B 0,C 180,E1 -5476.016,E2 -5476.016} C_VEL
LIN {X 0,Y 511.45,Z 237.687,A -85,B 0,C 180,E1 -5476.364,E2 -5476.364} C_VEL
LIN {X 0,Y 511.169,Z 249.871,A -85,B 0,C 180,E1 -5476.837,E2 -5476.837} C_VEL
LIN {X 0,Y 510.827,Z 261.536,A -85,B 0,C 180,E1 -5477.445,E2 -5477.445} C_VEL
LIN {X 0,Y 510.445,Z 272.505,A -85,B 0,C 180,E1 -5478.182,E2 -5478.182} C_VEL
LIN {X 0,Y 510.174,Z 283.204,A -85,B 0,C 180,E1 -5479.081,E2 -5479.081} C_VEL
LIN {X 0,Y 509.821,Z 292.847,A -85,B 0,C 180,E1 -5480.077,E2 -5480.077} C_VEL
LIN {X 0,Y 509.631,Z 300.762,A -85,B 0,C 180,E1 -5481.075,E2 -5481.075} C_VEL
LIN {X 0,Y 509.424,Z 308.492,A -85,B 0,C 180,E1 -5482.269,E2 -5482.269} C_VEL
LIN {X 0,Y 509.259,Z 315.62,A -85,B 0,C 180,E1 -5483.661,E2 -5483.661} C_VEL
LIN {X 0,Y 509.24,Z 320.367,A -85,B 0,C 180,E1 -5484.853,E2 -5484.853} C_VEL
LIN {X 0,Y 509.245,Z 323.995,A -85,B 0,C 180,E1 -5486.043,E2 -5486.043} C_VEL
LIN {X 0,Y 509.219,Z 325.866,A -85,B 0,C 180,E1 -5486.835,E2 -5486.835} C_VEL
LIN {X 0,Y 509.193,Z 327.269,A -85,B 0,C 180,E1 -5487.627,E2 -5487.627} C_VEL
LIN {X 0,Y 509.089,Z 328.88,A -85,B 0,C 180,E1 -5489.209,E2 -5489.209} C_VEL
LIN {X 0,Y 509.089,Z 329.099,A -85,B 0,C 180,E1 -5490,E2 -5490} C_VEL
LIN {X 0,Y 509.116,Z 328.278,A -85,B 0,C 180,E1 -5491.582,E2 -5491.582} C_VEL
LIN {X 0,Y 509.193,Z 327.284,A -85,B 0,C 180,E1 -5492.373,E2 -5492.373} C_VEL
LIN {X 0,Y 509.219,Z 325.885,A -85,B 0,C 180,E1 -5493.164,E2 -5493.164} C_VEL
LIN {X 0,Y 509.202,Z 322.939,A -85,B 0,C 180,E1 -5494.353,E2 -5494.353} C_VEL
LIN {X 0,Y 509.274,Z 318.954,A -85,B 0,C 180,E1 -5495.543,E2 -5495.543} C_VEL
LIN {X 0,Y 509.331,Z 312.923,A -85,B 0,C 180,E1 -5496.914,E2 -5496.914} C_VEL
LIN {X 0,Y 509.48,Z 306.124,A -85,B 0,C 180,E1 -5498.128,E2 -5498.128} C_VEL
LIN {X 0,Y 509.7,Z 297.815,A -85,B 0,C 180,E1 -5499.324,E2 -5499.324} C_VEL
LIN {X 0,Y 509.931,Z 289.3,A -85,B 0,C 180,E1 -5500.321,E2 -5500.321} C_VEL
LIN {X 0,Y 510.298,Z 278.784,A -85,B 0,C 180,E1 -5501.318,E2 -5501.318} C_VEL
LIN {X 0,Y 510.638,Z 267.044,A -85,B 0,C 180,E1 -5502.209,E2 -5502.209} C_VEL
LIN {X 0,Y 511,Z 255.037,A -85,B 0,C 180,E1 -5502.914,E2 -5502.914} C_VEL
LIN {X 0,Y 511.287,Z 242.65,A -85,B 0,C 180,E1 -5503.463,E2 -5503.463} C_VEL
LIN {X 0,Y 511.622,Z 229.933,A -85,B 0,C 180,E1 -5503.859,E2 -5503.859} C_VEL
LIN {X 0,Y 511.776,Z 214.795,A -85,B 0,C 180,E1 -5504.133,E2 -5504.133} C_VEL
LIN {X 0,Y 511.99,Z 128.414,A -85,B 0,C 180,E1 -5505.353,E2 -5505.353} C_VEL
LIN {X 0,Y 510.199,Z 115.809,A -85,B 0,C 180,E1 -5505.602,E2 -5505.602} C_VEL
LIN {X 0,Y 510.655,Z 95.735,A -85,B 0,C 180,E1 -5508.662,E2 -5508.662} C_VEL
LIN {X 0,Y 511.146,Z 76.776,A -85,B 0,C 180,E1 -5511.58,E2 -5511.58} C_VEL
LIN {X 0,Y 511.5,Z 63.191,A -85,B 0,C 180,E1 -5513.696,E2 -5513.696} C_VEL
LIN {X 0,Y 509.896,Z 53.972,A -85,B 0,C 180,E1 -5515.251,E2 -5515.251} C_VEL
LIN {X 0,Y 509.899,Z 53.971,A -85,B 0,C 180,E1 -5518.101,E2 -5518.101} C_VEL
LIN {X 0,Y 509.847,Z 53.972,A -85,B 0,C 180,E1 -5521.28,E2 -5521.28} C_VEL
LIN {X 0,Y 509.857,Z 53.974,A -85,B 0,C 180,E1 -5524.202,E2 -5524.202} C_VEL
LIN {X 0,Y 509.818,Z 53.978,A -85,B 0,C 180,E1 -5527.341,E2 -5527.341} C_VEL
LIN {X 0,Y 509.838,Z 53.973,A -85,B 0,C 180,E1 -5530.382,E2 -5530.382} C_VEL
LIN {X 0,Y 509.823,Z 53.977,A -85,B 0,C 180,E1 -5533.062,E2 -5533.062} C_VEL
LIN {X 0,Y 509.822,Z 53.979,A -85,B 0,C 180,E1 -5535.793,E2 -5535.793} C_VEL
LIN {X 0,Y 509.855,Z 53.971,A -85,B 0,C 180,E1 -5538.574,E2 -5538.574} C_VEL
LIN {X 0,Y 509.85,Z 53.973,A -85,B 0,C 180,E1 -5541.786,E2 -5541.786} C_VEL
LIN {X 0,Y 509.833,Z 53.975,A -85,B 0,C 180,E1 -5544.622,E2 -5544.622} C_VEL
LIN {X 0,Y 509.861,Z 53.973,A -85,B 0,C 180,E1 -5547.481,E2 -5547.481} C_VEL
LIN {X 0,Y 509.858,Z 53.971,A -85,B 0,C 180,E1 -5550.274,E2 -5550.274} C_VEL
LIN {X 0,Y 509.884,Z 53.976,A -85,B 0,C 180,E1 -5552.944,E2 -5552.944} C_VEL
LIN {X 0,Y 509.855,Z 53.971,A -85,B 0,C 180,E1 -5555.573,E2 -5555.573} C_VEL
LIN {X 0,Y 509.85,Z 53.976,A -85,B 0,C 180,E1 -5558.998,E2 -5558.998} C_VEL
LIN {X 0,Y 509.861,Z 53.97,A -85,B 0,C 180,E1 -5561.516,E2 -5561.516} C_VEL
LIN {X 0,Y 509.91,Z 53.969,A -85,B 0,C 180,E1 -5564.819,E2 -5564.819} C_VEL
LIN {X 0,Y 509.9,Z 53.969,A -85,B 0,C 180,E1 -5568.124,E2 -5568.124} C_VEL
LIN {X 0,Y 509.91,Z 53.964,A -85,B 0,C 180,E1 -5571.28,E2 -5571.28} C_VEL
LIN {X 0,Y 509.959,Z 53.959,A -85,B 0,C 180,E1 -5573.67,E2 -5573.67} C_VEL
LIN {X 0,Y 510.052,Z 53.948,A -85,B 0,C 180,E1 -5577.631,E2 -5577.631} C_VEL
LIN {X 0,Y 510.061,Z 53.945,A -85,B 0,C 180,E1 -5580.79,E2 -5580.79} C_VEL
LIN {X 0,Y 509.929,Z 53.961,A -85,B 0,C 180,E1 -5583.16,E2 -5583.16} C_VEL
LIN {X 0,Y 509.937,Z 53.963,A -85,B 0,C 180,E1 -5586.33,E2 -5586.33} C_VEL
LIN {X 0,Y 509.904,Z 53.964,A -85,B 0,C 180,E1 -5588.721,E2 -5588.721} C_VEL
LIN {X 0,Y 509.904,Z 53.97,A -85,B 0,C 180,E1 -5591.932,E2 -5591.932} C_VEL
LIN {X 0,Y 509.895,Z 53.969,A -85,B 0,C 180,E1 -5595.242,E2 -5595.242} C_VEL
LIN {X 0,Y 509.858,Z 53.97,A -85,B 0,C 180,E1 -5598.484,E2 -5598.484} C_VEL
LIN {X 0,Y 509.847,Z 53.974,A -85,B 0,C 180,E1 -5601.002,E2 -5601.002} C_VEL
LIN {X 0,Y 509.819,Z 53.98,A -85,B 0,C 180,E1 -5603.564,E2 -5603.564} C_VEL
LIN {X 0,Y 509.881,Z 53.967,A -85,B 0,C 180,E1 -5606.372,E2 -5606.372} C_VEL
LIN {X 0,Y 509.873,Z 53.972,A -85,B 0,C 180,E1 -5608.845,E2 -5608.845} C_VEL
LIN {X 0,Y 509.819,Z 53.977,A -85,B 0,C 180,E1 -5611.591,E2 -5611.591} C_VEL
LIN {X 0,Y 509.839,Z 53.974,A -85,B 0,C 180,E1 -5614.415,E2 -5614.415} C_VEL
LIN {X 0,Y 509.817,Z 53.978,A -85,B 0,C 180,E1 -5617.341,E2 -5617.341} C_VEL
LIN {X 0,Y 509.815,Z 53.978,A -85,B 0,C 180,E1 -5620.385,E2 -5620.385} C_VEL
LIN {X 0,Y 509.797,Z 53.982,A -85,B 0,C 180,E1 -5623.059,E2 -5623.059} C_VEL
LIN {X 0,Y 509.823,Z 53.974,A -85,B 0,C 180,E1 -5625.794,E2 -5625.794} C_VEL
LIN {X 0,Y 509.847,Z 53.98,A -85,B 0,C 180,E1 -5628.574,E2 -5628.574} C_VEL
LIN {X 0,Y 509.85,Z 53.972,A -85,B 0,C 180,E1 -5631.787,E2 -5631.787} C_VEL
LIN {X 0,Y 509.804,Z 53.977,A -85,B 0,C 180,E1 -5633.709,E2 -5633.709} C_VEL
LIN {X 0,Y 509.145,Z 54.068,A -85,B 0,C 180,E1 -5634.369,E2 -5634.369} C_VEL
LIN {X 0,Y 506.342,Z 54.411,A -85,B 0,C 180,E1 -5635.441,E2 -5635.441} C_VEL
LIN {X 0,Y 503.959,Z 54.714,A -85,B 0,C 180,E1 -5636.305,E2 -5636.305} C_VEL
LIN {X 0,Y 502.911,Z 54.837,A -85,B 0,C 180,E1 -5636.971,E2 -5636.971} C_VEL
LIN {X 0,Y 502.813,Z 54.848,A -85,B 0,C 180,E1 -5637.197,E2 -5637.197} C_VEL
LIN {X 0,Y 502.818,Z 54.854,A -85,B 0,C 180,E1 -5640.065,E2 -5640.065} C_VEL
LIN {X 0,Y 502.788,Z 54.854,A -85,B 0,C 180,E1 -5642.531,E2 -5642.531} C_VEL
LIN {X 0,Y 502.774,Z 54.853,A -85,B 0,C 180,E1 -5645.314,E2 -5645.314} C_VEL
LIN {X 0,Y 502.784,Z 54.858,A -85,B 0,C 180,E1 -5647.827,E2 -5647.827} C_VEL
LIN {X 0,Y 502.822,Z 54.848,A -85,B 0,C 180,E1 -5650.4,E2 -5650.4} C_VEL
LIN {X 0,Y 502.804,Z 54.849,A -85,B 0,C 180,E1 -5652.931,E2 -5652.931} C_VEL
LIN {X 0,Y 502.838,Z 54.853,A -85,B 0,C 180,E1 -5655.429,E2 -5655.429} C_VEL
LIN {X 0,Y 502.844,Z 54.936,A -85,B 0,C 180,E1 -5657.489,E2 -5657.489} C_VEL
LIN {X 0,Y 503.449,Z 58.849,A -85,B 0,C 180,E1 -5658.322,E2 -5658.322} C_VEL
LIN {X 0,Y 503.444,Z 70.777,A -85,B 0,C 180,E1 -5660.762,E2 -5660.762} C_VEL
LIN {X 0,Y 503.344,Z 73.357,A -85,B 0,C 180,E1 -5661.28,E2 -5661.28} C_VEL
LIN {X 0,Y 505.451,Z 84.676,A -85,B 0,C 180,E1 -5661.512,E2 -5661.512} C_VEL
LIN {X 0,Y 504.848,Z 179.61,A -85,B 0,C 180,E1 -5662.878,E2 -5662.878} C_VEL
LIN {X 0,Y 504.685,Z 192.791,A -85,B 0,C 180,E1 -5663.227,E2 -5663.227} C_VEL
LIN {X 0,Y 504.445,Z 205.966,A -85,B 0,C 180,E1 -5663.751,E2 -5663.751} C_VEL
LIN {X 0,Y 504.223,Z 217.828,A -85,B 0,C 180,E1 -5664.401,E2 -5664.401} C_VEL
LIN {X 0,Y 503.846,Z 229.177,A -85,B 0,C 180,E1 -5665.199,E2 -5665.199} C_VEL
LIN {X 0,Y 503.462,Z 239.416,A -85,B 0,C 180,E1 -5666.098,E2 -5666.098} C_VEL
LIN {X 0,Y 503.189,Z 247.792,A -85,B 0,C 180,E1 -5666.998,E2 -5666.998} C_VEL
LIN {X 0,Y 502.896,Z 255.537,A -85,B 0,C 180,E1 -5667.998,E2 -5667.998} C_VEL
LIN {X 0,Y 502.646,Z 263.116,A -85,B 0,C 180,E1 -5669.199,E2 -5669.199} C_VEL
LIN {X 0,Y 502.442,Z 269.215,A -85,B 0,C 180,E1 -5670.401,E2 -5670.401} C_VEL
LIN {X 0,Y 502.214,Z 274.079,A -85,B 0,C 180,E1 -5671.604,E2 -5671.604} C_VEL
LIN {X 0,Y 502.229,Z 277.826,A -85,B 0,C 180,E1 -5672.808,E2 -5672.808} C_VEL
LIN {X 0,Y 502.168,Z 280.578,A -85,B 0,C 180,E1 -5674.013,E2 -5674.013} C_VEL
LIN {X 0,Y 502.158,Z 282.79,A -85,B 0,C 180,E1 -5675.622,E2 -5675.622} C_VEL
LIN {X 0,Y 502.194,Z 283.315,A -85,B 0,C 180,E1 -5676.473,E2 -5676.473} C_VEL
LIN {X 0,Y 502.109,Z 283.101,A -85,B 0,C 180,E1 -5678.046,E2 -5678.046} C_VEL
LIN {X 0,Y 502.081,Z 282.42,A -85,B 0,C 180,E1 -5678.858,E2 -5678.858} C_VEL
LIN {X 0,Y 502.066,Z 281.329,A -85,B 0,C 180,E1 -5679.671,E2 -5679.671} C_VEL
LIN {X 0,Y 502.157,Z 279.783,A -85,B 0,C 180,E1 -5680.483,E2 -5680.483} C_VEL
LIN {X 0,Y 502.218,Z 276.999,A -85,B 0,C 180,E1 -5681.598,E2 -5681.598} C_VEL
LIN {X 0,Y 502.354,Z 272.455,A -85,B 0,C 180,E1 -5682.935,E2 -5682.935} C_VEL
LIN {X 0,Y 502.596,Z 266.006,A -85,B 0,C 180,E1 -5684.372,E2 -5684.372} C_VEL
LIN {X 0,Y 502.801,Z 258.898,A -85,B 0,C 180,E1 -5685.609,E2 -5685.609} C_VEL
LIN {X 0,Y 503.088,Z 249.944,A -85,B 0,C 180,E1 -5686.851,E2 -5686.851} C_VEL
LIN {X 0,Y 503.457,Z 240.715,A -85,B 0,C 180,E1 -5687.885,E2 -5687.885} C_VEL
LIN {X 0,Y 503.78,Z 230.394,A -85,B 0,C 180,E1 -5688.821,E2 -5688.821} C_VEL
LIN {X 0,Y 504.107,Z 218.837,A -85,B 0,C 180,E1 -5689.654,E2 -5689.654} C_VEL
LIN {X 0,Y 504.487,Z 206.767,A -85,B 0,C 180,E1 -5690.329,E2 -5690.329} C_VEL
LIN {X 0,Y 504.781,Z 194.239,A -85,B 0,C 180,E1 -5690.842,E2 -5690.842} C_VEL
LIN {X 0,Y 505.002,Z 180.745,A -85,B 0,C 180,E1 -5691.213,E2 -5691.213} C_VEL
LIN {X 0,Y 505.417,Z 107.413,A -85,B 0,C 180,E1 -5692.288,E2 -5692.288} C_VEL
LIN {X 0,Y 505.434,Z 83.316,A -85,B 0,C 180,E1 -5692.638,E2 -5692.638} C_VEL
LIN {X 0,Y 503.413,Z 73.415,A -85,B 0,C 180,E1 -5692.866,E2 -5692.866} C_VEL
LIN {X 0,Y 503.64,Z 59.97,A -85,B 0,C 180,E1 -5695.632,E2 -5695.632} C_VEL
LIN {X 0,Y 502.834,Z 54.853,A -85,B 0,C 180,E1 -5696.77,E2 -5696.77} C_VEL
LIN {X 0,Y 502.793,Z 54.859,A -85,B 0,C 180,E1 -5700.213,E2 -5700.213} C_VEL
LIN {X 0,Y 502.773,Z 54.856,A -85,B 0,C 180,E1 -5703.036,E2 -5703.036} C_VEL
LIN {X 0,Y 502.742,Z 54.864,A -85,B 0,C 180,E1 -5705.954,E2 -5705.954} C_VEL
LIN {X 0,Y 502.771,Z 54.855,A -85,B 0,C 180,E1 -5708.979,E2 -5708.979} C_VEL
LIN {X 0,Y 502.748,Z 54.861,A -85,B 0,C 180,E1 -5712.192,E2 -5712.192} C_VEL
LIN {X 0,Y 502.782,Z 54.851,A -85,B 0,C 180,E1 -5715.471,E2 -5715.471} C_VEL
LIN {X 0,Y 502.752,Z 54.855,A -85,B 0,C 180,E1 -5718.927,E2 -5718.927} C_VEL
LIN {X 0,Y 502.742,Z 54.859,A -85,B 0,C 180,E1 -5722.041,E2 -5722.041} C_VEL
LIN {X 0,Y 502.771,Z 54.855,A -85,B 0,C 180,E1 -5725.031,E2 -5725.031} C_VEL
LIN {X 0,Y 502.759,Z 54.854,A -85,B 0,C 180,E1 -5727.913,E2 -5727.913} C_VEL
LIN {X 0,Y 502.761,Z 54.857,A -85,B 0,C 180,E1 -5730.708,E2 -5730.708} C_VEL
LIN {X 0,Y 502.772,Z 54.857,A -85,B 0,C 180,E1 -5733.461,E2 -5733.461} C_VEL
LIN {X 0,Y 502.758,Z 54.854,A -85,B 0,C 180,E1 -5736.084,E2 -5736.084} C_VEL
LIN {X 0,Y 502.783,Z 54.855,A -85,B 0,C 180,E1 -5738.688,E2 -5738.688} C_VEL
LIN {X 0,Y 502.822,Z 54.848,A -85,B 0,C 180,E1 -5741.248,E2 -5741.248} C_VEL
LIN {X 0,Y 502.839,Z 54.852,A -85,B 0,C 180,E1 -5744.665,E2 -5744.665} C_VEL
LIN {X 0,Y 502.88,Z 54.837,A -85,B 0,C 180,E1 -5748.039,E2 -5748.039} C_VEL
LIN {X 0,Y 502.853,Z 54.844,A -85,B 0,C 180,E1 -5751.156,E2 -5751.156} C_VEL
LIN {X 0,Y 502.851,Z 54.84,A -85,B 0,C 180,E1 -5753.58,E2 -5753.58} C_VEL
LIN {X 0,Y 502.868,Z 54.844,A -85,B 0,C 180,E1 -5756.795,E2 -5756.795} C_VEL
LIN {X 0,Y 502.902,Z 54.84,A -85,B 0,C 180,E1 -5758.398,E2 -5758.398} C_VEL
LIN {X 0,Y 502.992,Z 54.825,A -85,B 0,C 180,E1 -5760.8,E2 -5760.8} C_VEL
LIN {X 0,Y 503.012,Z 54.828,A -85,B 0,C 180,E1 -5762.402,E2 -5762.402} C_VEL
LIN {X 0,Y 502.901,Z 54.838,A -85,B 0,C 180,E1 -5765.614,E2 -5765.614} C_VEL
LIN {X 0,Y 502.854,Z 54.849,A -85,B 0,C 180,E1 -5768.034,E2 -5768.034} C_VEL
LIN {X 0,Y 502.879,Z 54.839,A -85,B 0,C 180,E1 -5771.283,E2 -5771.283} C_VEL
LIN {X 0,Y 502.835,Z 54.845,A -85,B 0,C 180,E1 -5774.571,E2 -5774.571} C_VEL
LIN {X 0,Y 502.804,Z 54.851,A -85,B 0,C 180,E1 -5777.909,E2 -5777.909} C_VEL
LIN {X 0,Y 502.833,Z 54.845,A -85,B 0,C 180,E1 -5780.536,E2 -5780.536} C_VEL
LIN {X 0,Y 502.789,Z 54.851,A -85,B 0,C 180,E1 -5783.041,E2 -5783.041} C_VEL
LIN {X 0,Y 502.847,Z 54.843,A -85,B 0,C 180,E1 -5786.556,E2 -5786.556} C_VEL
LIN {X 0,Y 502.824,Z 54.853,A -85,B 0,C 180,E1 -5789.288,E2 -5789.288} C_VEL
LIN {X 0,Y 502.785,Z 54.851,A -85,B 0,C 180,E1 -5792.084,E2 -5792.084} C_VEL
LIN {X 0,Y 502.803,Z 54.851,A -85,B 0,C 180,E1 -5794.966,E2 -5794.966} C_VEL
LIN {X 0,Y 502.795,Z 54.847,A -85,B 0,C 180,E1 -5797.954,E2 -5797.954} C_VEL
LIN {X 0,Y 502.822,Z 54.851,A -85,B 0,C 180,E1 -5801.066,E2 -5801.066} C_VEL
LIN {X 0,Y 502.789,Z 54.859,A -85,B 0,C 180,E1 -5804.53,E2 -5804.53} C_VEL
LIN {X 0,Y 502.798,Z 54.851,A -85,B 0,C 180,E1 -5807.86,E2 -5807.86} C_VEL
LIN {X 0,Y 502.805,Z 54.85,A -85,B 0,C 180,E1 -5811.024,E2 -5811.024} C_VEL
LIN {X 0,Y 502.778,Z 54.857,A -85,B 0,C 180,E1 -5814.169,E2 -5814.169} C_VEL
LIN {X 0,Y 502.835,Z 54.849,A -85,B 0,C 180,E1 -5816.993,E2 -5816.993} C_VEL
LIN {X 0,Y 502.818,Z 54.857,A -85,B 0,C 180,E1 -5820.065,E2 -5820.065} C_VEL
LIN {X 0,Y 502.833,Z 54.85,A -85,B 0,C 180,E1 -5822.533,E2 -5822.533} C_VEL
LIN {X 0,Y 502.89,Z 54.984,A -85,B 0,C 180,E1 -5824.463,E2 -5824.463} C_VEL
LIN {X 0,Y 504.672,Z 64.891,A -85,B 0,C 180,E1 -5826.181,E2 -5826.181} C_VEL
LIN {X 0,Y 504.122,Z 82.981,A -85,B 0,C 180,E1 -5829.076,E2 -5829.076} C_VEL
LIN {X 0,Y 503.516,Z 103.658,A -85,B 0,C 180,E1 -5832.327,E2 -5832.327} C_VEL
LIN {X 0,Y 503.192,Z 115.487,A -85,B 0,C 180,E1 -5834.165,E2 -5834.165} C_VEL
LIN {X 0,Y 505.338,Z 131.554,A -85,B 0,C 180,E1 -5834.473,E2 -5834.473} C_VEL
LIN {X 0,Y 504.821,Z 224.422,A -85,B 0,C 180,E1 -5835.822,E2 -5835.822} C_VEL
LIN {X 0,Y 504.531,Z 237.58,A -85,B 0,C 180,E1 -5836.173,E2 -5836.173} C_VEL
LIN {X 0,Y 504.236,Z 249.692,A -85,B 0,C 180,E1 -5836.653,E2 -5836.653} C_VEL
LIN {X 0,Y 503.872,Z 261.86,A -85,B 0,C 180,E1 -5837.305,E2 -5837.305} C_VEL
LIN {X 0,Y 503.454,Z 273.534,A -85,B 0,C 180,E1 -5838.117,E2 -5838.117} C_VEL
LIN {X 0,Y 503.128,Z 283.991,A -85,B 0,C 180,E1 -5839.028,E2 -5839.028} C_VEL
LIN {X 0,Y 502.788,Z 292.545,A -85,B 0,C 180,E1 -5839.937,E2 -5839.937} C_VEL
LIN {X 0,Y 502.585,Z 300.447,A -85,B 0,C 180,E1 -5840.949,E2 -5840.949} C_VEL
LIN {X 0,Y 502.36,Z 308.172,A -85,B 0,C 180,E1 -5842.16,E2 -5842.16} C_VEL
LIN {X 0,Y 502.187,Z 315.298,A -85,B 0,C 180,E1 -5843.572,E2 -5843.572} C_VEL
LIN {X 0,Y 502.168,Z 320.045,A -85,B 0,C 180,E1 -5844.78,E2 -5844.78} C_VEL
LIN {X 0,Y 502.139,Z 323.672,A -85,B 0,C 180,E1 -5845.987,E2 -5845.987} C_VEL
LIN {X 0,Y 502.137,Z 325.544,A -85,B 0,C 180,E1 -5846.79,E2 -5846.79} C_VEL
LIN {X 0,Y 502.124,Z 326.948,A -85,B 0,C 180,E1 -5847.593,E2 -5847.593} C_VEL
LIN {X 0,Y 502.005,Z 328.559,A -85,B 0,C 180,E1 -5849.198,E2 -5849.198} C_VEL
LIN {X 0,Y 502.002,Z 328.779,A -85,B 0,C 180,E1 -5850,E2 -5850} C_VEL
LIN {X 0,Y 502.04,Z 327.959,A -85,B 0,C 180,E1 -5851.604,E2 -5851.604} C_VEL
LIN {X 0,Y 502.124,Z 326.965,A -85,B 0,C 180,E1 -5852.406,E2 -5852.406} C_VEL
LIN {X 0,Y 502.137,Z 325.566,A -85,B 0,C 180,E1 -5853.209,E2 -5853.209} C_VEL
LIN {X 0,Y 502.099,Z 322.619,A -85,B 0,C 180,E1 -5854.415,E2 -5854.415} C_VEL
LIN {X 0,Y 502.185,Z 318.633,A -85,B 0,C 180,E1 -5855.622,E2 -5855.622} C_VEL
LIN {X 0,Y 502.272,Z 312.6,A -85,B 0,C 180,E1 -5857.012,E2 -5857.012} C_VEL
LIN {X 0,Y 502.418,Z 305.796,A -85,B 0,C 180,E1 -5858.243,E2 -5858.243} C_VEL
LIN {X 0,Y 502.656,Z 297.483,A -85,B 0,C 180,E1 -5859.455,E2 -5859.455} C_VEL
LIN {X 0,Y 502.929,Z 288.957,A -85,B 0,C 180,E1 -5860.466,E2 -5860.466} C_VEL
LIN {X 0,Y 503.299,Z 278.42,A -85,B 0,C 180,E1 -5861.477,E2 -5861.477} C_VEL
LIN {X 0,Y 503.656,Z 266.802,A -85,B 0,C 180,E1 -5862.371,E2 -5862.371} C_VEL
LIN {X 0,Y 504.04,Z 254.614,A -85,B 0,C 180,E1 -5863.096,E2 -5863.096} C_VEL
LIN {X 0,Y 504.379,Z 242.184,A -85,B 0,C 180,E1 -5863.651,E2 -5863.651} C_VEL
LIN {X 0,Y 504.725,Z 229.37,A -85,B 0,C 180,E1 -5864.052,E2 -5864.052} C_VEL
LIN {X 0,Y 504.874,Z 215.777,A -85,B 0,C 180,E1 -5864.305,E2 -5864.305} C_VEL
LIN {X 0,Y 505.154,Z 129.397,A -85,B 0,C 180,E1 -5865.539,E2 -5865.539} C_VEL
LIN {X 0,Y 503.199,Z 115.466,A -85,B 0,C 180,E1 -5865.819,E2 -5865.819} C_VEL
LIN {X 0,Y 503.737,Z 93.984,A -85,B 0,C 180,E1 -5869.139,E2 -5869.139} C_VEL
LIN {X 0,Y 504.218,Z 75.001,A -85,B 0,C 180,E1 -5872.107,E2 -5872.107} C_VEL
LIN {X 0,Y 504.526,Z 64.123,A -85,B 0,C 180,E1 -5873.826,E2 -5873.826} C_VEL
LIN {X 0,Y 502.849,Z 54.85,A -85,B 0,C 180,E1 -5875.397,E2 -5875.397} C_VEL
LIN {X 0,Y 502.842,Z 54.851,A -85,B 0,C 180,E1 -5878.372,E2 -5878.372} C_VEL
LIN {X 0,Y 502.794,Z 54.853,A -85,B 0,C 180,E1 -5881.499,E2 -5881.499} C_VEL
LIN {X 0,Y 502.805,Z 54.855,A -85,B 0,C 180,E1 -5883.994,E2 -5883.994} C_VEL
LIN {X 0,Y 502.778,Z 54.854,A -85,B 0,C 180,E1 -5887.178,E2 -5887.178} C_VEL
LIN {X 0,Y 502.788,Z 54.855,A -85,B 0,C 180,E1 -5890.015,E2 -5890.015} C_VEL
LIN {X 0,Y 502.803,Z 54.85,A -85,B 0,C 180,E1 -5892.199,E2 -5892.199} C_VEL
LIN {X 0,Y 502.786,Z 54.859,A -85,B 0,C 180,E1 -5895.47,E2 -5895.47} C_VEL
LIN {X 0,Y 502.819,Z 54.85,A -85,B 0,C 180,E1 -5898.934,E2 -5898.934} C_VEL
LIN {X 0,Y 502.792,Z 54.851,A -85,B 0,C 180,E1 -5902.046,E2 -5902.046} C_VEL
LIN {X 0,Y 502.802,Z 54.855,A -85,B 0,C 180,E1 -5905.034,E2 -5905.034} C_VEL
LIN {X 0,Y 502.783,Z 54.852,A -85,B 0,C 180,E1 -5907.915,E2 -5907.915} C_VEL
LIN {X 0,Y 502.823,Z 54.851,A -85,B 0,C 180,E1 -5910.712,E2 -5910.712} C_VEL
LIN {X 0,Y 502.862,Z 54.844,A -85,B 0,C 180,E1 -5913.439,E2 -5913.439} C_VEL
LIN {X 0,Y 502.776,Z 54.853,A -85,B 0,C 180,E1 -5916.086,E2 -5916.086} C_VEL
LIN {X 0,Y 502.783,Z 54.859,A -85,B 0,C 180,E1 -5918.689,E2 -5918.689} C_VEL
LIN {X 0,Y 502.826,Z 54.848,A -85,B 0,C 180,E1 -5921.248,E2 -5921.248} C_VEL
LIN {X 0,Y 502.848,Z 54.852,A -85,B 0,C 180,E1 -5924.6,E2 -5924.6} C_VEL
LIN {X 0,Y 502.876,Z 54.843,A -85,B 0,C 180,E1 -5928.039,E2 -5928.039} C_VEL
LIN {X 0,Y 502.869,Z 54.841,A -85,B 0,C 180,E1 -5931.157,E2 -5931.157} C_VEL
LIN {X 0,Y 502.911,Z 54.836,A -85,B 0,C 180,E1 -5933.581,E2 -5933.581} C_VEL
LIN {X 0,Y 502.873,Z 54.842,A -85,B 0,C 180,E1 -5936.795,E2 -5936.795} C_VEL
LIN {X 0,Y 502.896,Z 54.842,A -85,B 0,C 180,E1 -5938.399,E2 -5938.399} C_VEL
LIN {X 0,Y 503.011,Z 54.824,A -85,B 0,C 180,E1 -5940.801,E2 -5940.801} C_VEL
LIN {X 0,Y 502.874,Z 54.84,A -85,B 0,C 180,E1 -5943.205,E2 -5943.205} C_VEL
LIN {X 0,Y 502.887,Z 54.84,A -85,B 0,C 180,E1 -5946.419,E2 -5946.419} C_VEL
LIN {X 0,Y 502.864,Z 54.841,A -85,B 0,C 180,E1 -5948.844,E2 -5948.844} C_VEL
LIN {X 0,Y 502.845,Z 54.847,A -85,B 0,C 180,E1 -5952.102,E2 -5952.102} C_VEL
LIN {X 0,Y 502.849,Z 54.849,A -85,B 0,C 180,E1 -5955.4,E2 -5955.4} C_VEL
LIN {X 0,Y 502.823,Z 54.847,A -85,B 0,C 180,E1 -5958.752,E2 -5958.752} C_VEL
LIN {X 0,Y 502.781,Z 54.859,A -85,B 0,C 180,E1 -5961.312,E2 -5961.312} C_VEL
LIN {X 0,Y 502.769,Z 54.855,A -85,B 0,C 180,E1 -5963.915,E2 -5963.915} C_VEL
LIN {X 0,Y 502.836,Z 54.846,A -85,B 0,C 180,E1 -5966.568,E2 -5966.568} C_VEL
LIN {X 0,Y 502.823,Z 54.853,A -85,B 0,C 180,E1 -5969.288,E2 -5969.288} C_VEL
LIN {X 0,Y 502.783,Z 54.851,A -85,B 0,C 180,E1 -5972.085,E2 -5972.085} C_VEL
LIN {X 0,Y 502.796,Z 54.858,A -85,B 0,C 180,E1 -5974.967,E2 -5974.967} C_VEL
LIN {X 0,Y 502.793,Z 54.85,A -85,B 0,C 180,E1 -5977.954,E2 -5977.954} C_VEL
LIN {X 0,Y 502.772,Z 54.857,A -85,B 0,C 180,E1 -5981.071,E2 -5981.071} C_VEL
LIN {X 0,Y 502.78,Z 54.855,A -85,B 0,C 180,E1 -5984.341,E2 -5984.341} C_VEL
LIN {X 0,Y 502.76,Z 54.861,A -85,B 0,C 180,E1 -5986.768,E2 -5986.768} C_VEL
LIN {X 0,Y 502.796,Z 54.852,A -85,B 0,C 180,E1 -5989.009,E2 -5989.009} C_VEL
LIN {X 0,Y 502.79,Z 54.854,A -85,B 0,C 180,E1 -5992.046,E2 -5992.046} C_VEL
LIN {X 0,Y 502.796,Z 54.851,A -85,B 0,C 180,E1 -5995.034,E2 -5995.034} C_VEL
LIN {X 0,Y 502.813,Z 54.848,A -85,B 0,C 180,E1 -5997.197,E2 -5997.197} C_VEL
LIN {X 0,Y 502.111,Z 54.94,A -85,B 0,C 180,E1 -5997.865,E2 -5997.865} C_VEL
LIN {X 0,Y 499.25,Z 55.296,A -85,B 0,C 180,E1 -5998.951,E2 -5998.951} C_VEL
LIN {X 0,Y 496.853,Z 55.596,A -85,B 0,C 180,E1 -5999.826,E2 -5999.826} C_VEL
LIN {X 0,Y 495.824,Z 55.723,A -85,B 0,C 180,E1 -6000.502,E2 -6000.502} C_VEL
LIN {X 0,Y 495.74,Z 55.731,A -85,B 0,C 180,E1 -6000.73,E2 -6000.73} C_VEL
LIN {X 0,Y 495.72,Z 55.738,A -85,B 0,C 180,E1 -6003.928,E2 -6003.928} C_VEL
LIN {X 0,Y 495.762,Z 55.726,A -85,B 0,C 180,E1 -6007.14,E2 -6007.14} C_VEL
LIN {X 0,Y 495.771,Z 55.73,A -85,B 0,C 180,E1 -6010.11,E2 -6010.11} C_VEL
LIN {X 0,Y 495.748,Z 55.728,A -85,B 0,C 180,E1 -6012.68,E2 -6012.68} C_VEL
LIN {X 0,Y 495.787,Z 55.729,A -85,B 0,C 180,E1 -6015.217,E2 -6015.217} C_VEL
LIN {X 0,Y 495.816,Z 55.806,A -85,B 0,C 180,E1 -6017.36,E2 -6017.36} C_VEL
LIN {X 0,Y 496.486,Z 61.47,A -85,B 0,C 180,E1 -6018.57,E2 -6018.57} C_VEL
LIN {X 0,Y 496.388,Z 73.594,A -85,B 0,C 180,E1 -6021.06,E2 -6021.06} C_VEL
LIN {X 0,Y 498.602,Z 85.57,A -85,B 0,C 180,E1 -6021.316,E2 -6021.316} C_VEL
LIN {X 0,Y 497.945,Z 180.454,A -85,B 0,C 180,E1 -6022.702,E2 -6022.702} C_VEL
LIN {X 0,Y 497.773,Z 194.204,A -85,B 0,C 180,E1 -6023.082,E2 -6023.082} C_VEL
LIN {X 0,Y 497.536,Z 205.992,A -85,B 0,C 180,E1 -6023.563,E2 -6023.563} C_VEL
LIN {X 0,Y 497.306,Z 217.945,A -85,B 0,C 180,E1 -6024.221,E2 -6024.221} C_VEL
LIN {X 0,Y 496.875,Z 229.342,A -85,B 0,C 180,E1 -6025.03,E2 -6025.03} C_VEL
LIN {X 0,Y 496.486,Z 239.61,A -85,B 0,C 180,E1 -6025.942,E2 -6025.942} C_VEL
LIN {X 0,Y 496.165,Z 248.868,A -85,B 0,C 180,E1 -6026.955,E2 -6026.955} C_VEL
LIN {X 0,Y 495.807,Z 257.814,A -85,B 0,C 180,E1 -6028.173,E2 -6028.173} C_VEL
LIN {X 0,Y 495.595,Z 265.029,A -85,B 0,C 180,E1 -6029.391,E2 -6029.391} C_VEL
LIN {X 0,Y 495.24,Z 271.68,A -85,B 0,C 180,E1 -6030.813,E2 -6030.813} C_VEL
LIN {X 0,Y 495.178,Z 276.065,A -85,B 0,C 180,E1 -6032.034,E2 -6032.034} C_VEL
LIN {X 0,Y 495.142,Z 279.4,A -85,B 0,C 180,E1 -6033.255,E2 -6033.255} C_VEL
LIN {X 0,Y 495.082,Z 281.063,A -85,B 0,C 180,E1 -6034.07,E2 -6034.07} C_VEL
LIN {X 0,Y 495.077,Z 283.201,A -85,B 0,C 180,E1 -6035.703,E2 -6035.703} C_VEL
LIN {X 0,Y 495.108,Z 283.645,A -85,B 0,C 180,E1 -6036.521,E2 -6036.521} C_VEL
LIN {X 0,Y 495.012,Z 283.367,A -85,B 0,C 180,E1 -6038.162,E2 -6038.162} C_VEL
LIN {X 0,Y 495.011,Z 282.647,A -85,B 0,C 180,E1 -6038.985,E2 -6038.985} C_VEL
LIN {X 0,Y 494.996,Z 281.484,A -85,B 0,C 180,E1 -6039.81,E2 -6039.81} C_VEL
LIN {X 0,Y 495.12,Z 278.964,A -85,B 0,C 180,E1 -6041.048,E2 -6041.048} C_VEL
LIN {X 0,Y 495.258,Z 275.416,A -85,B 0,C 180,E1 -6042.29,E2 -6042.29} C_VEL
LIN {X 0,Y 495.352,Z 270.723,A -85,B 0,C 180,E1 -6043.539,E2 -6043.539} C_VEL
LIN {X 0,Y 495.605,Z 264.738,A -85,B 0,C 180,E1 -6044.789,E2 -6044.789} C_VEL
LIN {X 0,Y 495.851,Z 257.235,A -85,B 0,C 180,E1 -6046.045,E2 -6046.045} C_VEL
LIN {X 0,Y 496.131,Z 249.536,A -85,B 0,C 180,E1 -6047.094,E2 -6047.094} C_VEL
LIN {X 0,Y 496.542,Z 240.131,A -85,B 0,C 180,E1 -6048.143,E2 -6048.143} C_VEL
LIN {X 0,Y 496.892,Z 229.565,A -85,B 0,C 180,E1 -6049.092,E2 -6049.092} C_VEL
LIN {X 0,Y 497.283,Z 217.764,A -85,B 0,C 180,E1 -6049.935,E2 -6049.935} C_VEL
LIN {X 0,Y 497.672,Z 206.295,A -85,B 0,C 180,E1 -6050.566,E2 -6050.566} C_VEL
LIN {X 0,Y 497.924,Z 193.16,A -85,B 0,C 180,E1 -6051.098,E2 -6051.098} C_VEL
LIN {X 0,Y 498.185,Z 179.628,A -85,B 0,C 180,E1 -6051.457,E2 -6051.457} C_VEL
LIN {X 0,Y 498.616,Z 84.179,A -85,B 0,C 180,E1 -6052.865,E2 -6052.865} C_VEL
LIN {X 0,Y 496.469,Z 73.674,A -85,B 0,C 180,E1 -6053.119,E2 -6053.119} C_VEL
LIN {X 0,Y 496.74,Z 61.885,A -85,B 0,C 180,E1 -6055.564,E2 -6055.564} C_VEL
LIN {X 0,Y 495.799,Z 55.729,A -85,B 0,C 180,E1 -6056.936,E2 -6056.936} C_VEL
LIN {X 0,Y 495.748,Z 55.736,A -85,B 0,C 180,E1 -6060.143,E2 -6060.143} C_VEL
LIN {X 0,Y 495.731,Z 55.733,A -85,B 0,C 180,E1 -6063.233,E2 -6063.233} C_VEL
LIN {X 0,Y 495.685,Z 55.746,A -85,B 0,C 180,E1 -6066.082,E2 -6066.082} C_VEL
LIN {X 0,Y 495.732,Z 55.732,A -85,B 0,C 180,E1 -6068.763,E2 -6068.763} C_VEL
LIN {X 0,Y 495.703,Z 55.74,A -85,B 0,C 180,E1 -6071.787,E2 -6071.787} C_VEL
LIN {X 0,Y 495.735,Z 55.725,A -85,B 0,C 180,E1 -6075.142,E2 -6075.142} C_VEL
LIN {X 0,Y 495.704,Z 55.734,A -85,B 0,C 180,E1 -6078.213,E2 -6078.213} C_VEL
LIN {X 0,Y 495.706,Z 55.739,A -85,B 0,C 180,E1 -6081.404,E2 -6081.404} C_VEL
LIN {X 0,Y 495.721,Z 55.73,A -85,B 0,C 180,E1 -6084.46,E2 -6084.46} C_VEL
LIN {X 0,Y 495.727,Z 55.736,A -85,B 0,C 180,E1 -6087.402,E2 -6087.402} C_VEL
LIN {X 0,Y 495.703,Z 55.734,A -85,B 0,C 180,E1 -6090.249,E2 -6090.249} C_VEL
LIN {X 0,Y 495.723,Z 55.737,A -85,B 0,C 180,E1 -6093.275,E2 -6093.275} C_VEL
LIN {X 0,Y 495.706,Z 55.734,A -85,B 0,C 180,E1 -6095.722,E2 -6095.722} C_VEL
LIN {X 0,Y 495.743,Z 55.728,A -85,B 0,C 180,E1 -6098.371,E2 -6098.371} C_VEL
LIN {X 0,Y 495.777,Z 55.729,A -85,B 0,C 180,E1 -6100.971,E2 -6100.971} C_VEL
LIN {X 0,Y 495.825,Z 55.723,A -85,B 0,C 180,E1 -6104.549,E2 -6104.549} C_VEL
LIN {X 0,Y 495.832,Z 55.715,A -85,B 0,C 180,E1 -6107.965,E2 -6107.965} C_VEL
LIN {X 0,Y 495.81,Z 55.722,A -85,B 0,C 180,E1 -6111.029,E2 -6111.029} C_VEL
LIN {X 0,Y 495.807,Z 55.717,A -85,B 0,C 180,E1 -6113.488,E2 -6113.488} C_VEL
LIN {X 0,Y 495.723,Z 55.733,A -85,B 0,C 180,E1 -6115.935,E2 -6115.935} C_VEL
LIN {X 0,Y 495.985,Z 55.7,A -85,B 0,C 180,E1 -6117.563,E2 -6117.563} C_VEL
LIN {X 0,Y 495.944,Z 55.703,A -85,B 0,C 180,E1 -6120.812,E2 -6120.812} C_VEL
LIN {X 0,Y 495.979,Z 55.703,A -85,B 0,C 180,E1 -6122.436,E2 -6122.436} C_VEL
LIN {X 0,Y 495.859,Z 55.716,A -85,B 0,C 180,E1 -6125.694,E2 -6125.694} C_VEL
LIN {X 0,Y 495.818,Z 55.724,A -85,B 0,C 180,E1 -6128.149,E2 -6128.149} C_VEL
LIN {X 0,Y 495.854,Z 55.716,A -85,B 0,C 180,E1 -6131.445,E2 -6131.445} C_VEL
LIN {X 0,Y 495.783,Z 55.724,A -85,B 0,C 180,E1 -6134.783,E2 -6134.783} C_VEL
LIN {X 0,Y 495.775,Z 55.724,A -85,B 0,C 180,E1 -6138.234,E2 -6138.234} C_VEL
LIN {X 0,Y 495.777,Z 55.725,A -85,B 0,C 180,E1 -6140.756,E2 -6140.756} C_VEL
LIN {X 0,Y 495.742,Z 55.734,A -85,B 0,C 180,E1 -6143.387,E2 -6143.387} C_VEL
LIN {X 0,Y 495.808,Z 55.721,A -85,B 0,C 180,E1 -6146.745,E2 -6146.745} C_VEL
LIN {X 0,Y 495.767,Z 55.726,A -85,B 0,C 180,E1 -6149.746,E2 -6149.746} C_VEL
LIN {X 0,Y 495.77,Z 55.728,A -85,B 0,C 180,E1 -6152.594,E2 -6152.594} C_VEL
LIN {X 0,Y 495.752,Z 55.721,A -85,B 0,C 180,E1 -6155.537,E2 -6155.537} C_VEL
LIN {X 0,Y 495.765,Z 55.731,A -85,B 0,C 180,E1 -6158.768,E2 -6158.768} C_VEL
LIN {X 0,Y 495.759,Z 55.727,A -85,B 0,C 180,E1 -6161.781,E2 -6161.781} C_VEL
LIN {X 0,Y 495.74,Z 55.731,A -85,B 0,C 180,E1 -6165.141,E2 -6165.141} C_VEL
LIN {X 0,Y 495.759,Z 55.731,A -85,B 0,C 180,E1 -6168.219,E2 -6168.219} C_VEL
LIN {X 0,Y 495.753,Z 55.728,A -85,B 0,C 180,E1 -6171.408,E2 -6171.408} C_VEL
LIN {X 0,Y 495.751,Z 55.731,A -85,B 0,C 180,E1 -6174.462,E2 -6174.462} C_VEL
LIN {X 0,Y 495.77,Z 55.73,A -85,B 0,C 180,E1 -6177.406,E2 -6177.406} C_VEL
LIN {X 0,Y 495.769,Z 55.734,A -85,B 0,C 180,E1 -6180.254,E2 -6180.254} C_VEL
LIN {X 0,Y 495.826,Z 55.723,A -85,B 0,C 180,E1 -6183.251,E2 -6183.251} C_VEL
LIN {X 0,Y 495.835,Z 55.857,A -85,B 0,C 180,E1 -6184.245,E2 -6184.245} C_VEL
LIN {X 0,Y 497.758,Z 66.208,A -85,B 0,C 180,E1 -6186.072,E2 -6186.072} C_VEL
LIN {X 0,Y 497.165,Z 84.399,A -85,B 0,C 180,E1 -6189.029,E2 -6189.029} C_VEL
LIN {X 0,Y 496.513,Z 104.782,A -85,B 0,C 180,E1 -6192.282,E2 -6192.282} C_VEL
LIN {X 0,Y 496.201,Z 115.221,A -85,B 0,C 180,E1 -6193.925,E2 -6193.925} C_VEL
LIN {X 0,Y 498.511,Z 131.664,A -85,B 0,C 180,E1 -6194.248,E2 -6194.248} C_VEL
LIN {X 0,Y 498.005,Z 223.474,A -85,B 0,C 180,E1 -6195.597,E2 -6195.597} C_VEL
LIN {X 0,Y 497.69,Z 236.838,A -85,B 0,C 180,E1 -6195.953,E2 -6195.953} C_VEL
LIN {X 0,Y 497.304,Z 249.613,A -85,B 0,C 180,E1 -6196.463,E2 -6196.463} C_VEL
LIN {X 0,Y 496.912,Z 262.004,A -85,B 0,C 180,E1 -6197.144,E2 -6197.144} C_VEL
LIN {X 0,Y 496.454,Z 273.33,A -85,B 0,C 180,E1 -6197.947,E2 -6197.947} C_VEL
LIN {X 0,Y 496.103,Z 283.755,A -85,B 0,C 180,E1 -6198.871,E2 -6198.871} C_VEL
LIN {X 0,Y 495.757,Z 292.289,A -85,B 0,C 180,E1 -6199.793,E2 -6199.793} C_VEL
LIN {X 0,Y 495.49,Z 301.553,A -85,B 0,C 180,E1 -6201.024,E2 -6201.024} C_VEL
LIN {X 0,Y 495.254,Z 309.003,A -85,B 0,C 180,E1 -6202.252,E2 -6202.252} C_VEL
LIN {X 0,Y 495.088,Z 315.343,A -85,B 0,C 180,E1 -6203.557,E2 -6203.557} C_VEL
LIN {X 0,Y 495.097,Z 319.736,A -85,B 0,C 180,E1 -6204.706,E2 -6204.706} C_VEL
LIN {X 0,Y 495.033,Z 323.357,A -85,B 0,C 180,E1 -6205.929,E2 -6205.929} C_VEL
LIN {X 0,Y 495.056,Z 325.229,A -85,B 0,C 180,E1 -6206.744,E2 -6206.744} C_VEL
LIN {X 0,Y 495.028,Z 326.63,A -85,B 0,C 180,E1 -6207.559,E2 -6207.559} C_VEL
LIN {X 0,Y 494.924,Z 328.241,A -85,B 0,C 180,E1 -6209.186,E2 -6209.186} C_VEL
LIN {X 0,Y 494.918,Z 328.459,A -85,B 0,C 180,E1 -6210,E2 -6210} C_VEL
LIN {X 0,Y 494.966,Z 327.637,A -85,B 0,C 180,E1 -6211.627,E2 -6211.627} C_VEL
LIN {X 0,Y 495.028,Z 326.642,A -85,B 0,C 180,E1 -6212.441,E2 -6212.441} C_VEL
LIN {X 0,Y 495.056,Z 325.241,A -85,B 0,C 180,E1 -6213.255,E2 -6213.255} C_VEL
LIN {X 0,Y 495.005,Z 322.29,A -85,B 0,C 180,E1 -6214.478,E2 -6214.478} C_VEL
LIN {X 0,Y 495.077,Z 318.298,A -85,B 0,C 180,E1 -6215.703,E2 -6215.703} C_VEL
LIN {X 0,Y 495.202,Z 312.155,A -85,B 0,C 180,E1 -6217.133,E2 -6217.133} C_VEL
LIN {X 0,Y 495.346,Z 305.442,A -85,B 0,C 180,E1 -6218.362,E2 -6218.362} C_VEL
LIN {X 0,Y 495.616,Z 297.112,A -85,B 0,C 180,E1 -6219.591,E2 -6219.591} C_VEL
LIN {X 0,Y 495.905,Z 288.562,A -85,B 0,C 180,E1 -6220.616,E2 -6220.616} C_VEL
LIN {X 0,Y 496.309,Z 278.001,A -85,B 0,C 180,E1 -6221.641,E2 -6221.641} C_VEL
LIN {X 0,Y 496.676,Z 266.573,A -85,B 0,C 180,E1 -6222.532,E2 -6222.532} C_VEL
LIN {X 0,Y 497.1,Z 254.098,A -85,B 0,C 180,E1 -6223.282,E2 -6223.282} C_VEL
LIN {X 0,Y 497.46,Z 241.588,A -85,B 0,C 180,E1 -6223.844,E2 -6223.844} C_VEL
LIN {X 0,Y 497.849,Z 228.602,A -85,B 0,C 180,E1 -6224.25,E2 -6224.25} C_VEL
LIN {X 0,Y 497.982,Z 212.871,A -85,B 0,C 180,E1 -6224.533,E2 -6224.533} C_VEL
LIN {X 0,Y 498.319,Z 130.248,A -85,B 0,C 180,E1 -6225.728,E2 -6225.728} C_VEL
LIN {X 0,Y 496.164,Z 115.134,A -85,B 0,C 180,E1 -6226.037,E2 -6226.037} C_VEL
LIN {X 0,Y 496.719,Z 94.914,A -85,B 0,C 180,E1 -6229.205,E2 -6229.205} C_VEL
LIN {X 0,Y 497.188,Z 77.281,A -85,B 0,C 180,E1 -6231.999,E2 -6231.999} C_VEL
LIN {X 0,Y 497.534,Z 65.042,A -85,B 0,C 180,E1 -6233.96,E2 -6233.96} C_VEL
LIN {X 0,Y 495.803,Z 55.728,A -85,B 0,C 180,E1 -6235.559,E2 -6235.559} C_VEL
LIN {X 0,Y 495.789,Z 55.728,A -85,B 0,C 180,E1 -6238.493,E2 -6238.493} C_VEL
LIN {X 0,Y 495.756,Z 55.732,A -85,B 0,C 180,E1 -6241.725,E2 -6241.725} C_VEL
LIN {X 0,Y 495.769,Z 55.725,A -85,B 0,C 180,E1 -6244.694,E2 -6244.694} C_VEL
LIN {X 0,Y 495.73,Z 55.736,A -85,B 0,C 180,E1 -6247.561,E2 -6247.561} C_VEL
LIN {X 0,Y 495.766,Z 55.725,A -85,B 0,C 180,E1 -6250.7,E2 -6250.7} C_VEL
LIN {X 0,Y 495.727,Z 55.733,A -85,B 0,C 180,E1 -6254.001,E2 -6254.001} C_VEL
LIN {X 0,Y 495.725,Z 55.735,A -85,B 0,C 180,E1 -6257.117,E2 -6257.117} C_VEL
LIN {X 0,Y 495.758,Z 55.728,A -85,B 0,C 180,E1 -6259.953,E2 -6259.953} C_VEL
LIN {X 0,Y 495.727,Z 55.731,A -85,B 0,C 180,E1 -6262.553,E2 -6262.553} C_VEL
LIN {X 0,Y 495.781,Z 55.728,A -85,B 0,C 180,E1 -6265.457,E2 -6265.457} C_VEL
LIN {X 0,Y 495.755,Z 55.728,A -85,B 0,C 180,E1 -6268.364,E2 -6268.364} C_VEL
LIN {X 0,Y 495.786,Z 55.725,A -85,B 0,C 180,E1 -6271.507,E2 -6271.507} C_VEL
LIN {X 0,Y 495.789,Z 55.723,A -85,B 0,C 180,E1 -6273.932,E2 -6273.932} C_VEL
LIN {X 0,Y 495.758,Z 55.73,A -85,B 0,C 180,E1 -6277.14,E2 -6277.14} C_VEL
LIN {X 0,Y 495.77,Z 55.726,A -85,B 0,C 180,E1 -6280.11,E2 -6280.11} C_VEL
LIN {X 0,Y 495.763,Z 55.734,A -85,B 0,C 180,E1 -6282.681,E2 -6282.681} C_VEL
LIN {X 0,Y 495.788,Z 55.724,A -85,B 0,C 180,E1 -6285.217,E2 -6285.217} C_VEL
LIN {X 0,Y 495.851,Z 55.722,A -85,B 0,C 180,E1 -6288.555,E2 -6288.555} C_VEL
LIN {X 0,Y 495.871,Z 55.715,A -85,B 0,C 180,E1 -6291.852,E2 -6291.852} C_VEL
LIN {X 0,Y 495.889,Z 55.718,A -85,B 0,C 180,E1 -6294.307,E2 -6294.307} C_VEL
LIN {X 0,Y 495.988,Z 55.699,A -85,B 0,C 180,E1 -6297.564,E2 -6297.564} C_VEL
LIN {X 0,Y 495.962,Z 55.702,A -85,B 0,C 180,E1 -6300.812,E2 -6300.812} C_VEL
LIN {X 0,Y 495.988,Z 55.701,A -85,B 0,C 180,E1 -6302.437,E2 -6302.437} C_VEL
LIN {X 0,Y 495.881,Z 55.717,A -85,B 0,C 180,E1 -6305.694,E2 -6305.694} C_VEL
LIN {X 0,Y 495.834,Z 55.717,A -85,B 0,C 180,E1 -6308.97,E2 -6308.97} C_VEL
LIN {X 0,Y 495.829,Z 55.722,A -85,B 0,C 180,E1 -6312.035,E2 -6312.035} C_VEL
LIN {X 0,Y 495.824,Z 55.725,A -85,B 0,C 180,E1 -6315.452,E2 -6315.452} C_VEL
LIN {X 0,Y 495.779,Z 55.726,A -85,B 0,C 180,E1 -6319.029,E2 -6319.029} C_VEL
LIN {X 0,Y 495.741,Z 55.734,A -85,B 0,C 180,E1 -6321.629,E2 -6321.629} C_VEL
LIN {X 0,Y 495.716,Z 55.732,A -85,B 0,C 180,E1 -6324.277,E2 -6324.277} C_VEL
LIN {X 0,Y 495.784,Z 55.728,A -85,B 0,C 180,E1 -6326.976,E2 -6326.976} C_VEL
LIN {X 0,Y 495.766,Z 55.727,A -85,B 0,C 180,E1 -6329.747,E2 -6329.747} C_VEL
LIN {X 0,Y 495.767,Z 55.728,A -85,B 0,C 180,E1 -6332.595,E2 -6332.595} C_VEL
LIN {X 0,Y 495.748,Z 55.729,A -85,B 0,C 180,E1 -6335.538,E2 -6335.538} C_VEL
LIN {X 0,Y 495.759,Z 55.734,A -85,B 0,C 180,E1 -6338.768,E2 -6338.768} C_VEL
LIN {X 0,Y 495.735,Z 55.729,A -85,B 0,C 180,E1 -6341.784,E2 -6341.784} C_VEL
LIN {X 0,Y 495.739,Z 55.731,A -85,B 0,C 180,E1 -6345.141,E2 -6345.141} C_VEL
LIN {X 0,Y 495.751,Z 55.731,A -85,B 0,C 180,E1 -6348.219,E2 -6348.219} C_VEL
LIN {X 0,Y 495.749,Z 55.728,A -85,B 0,C 180,E1 -6351.409,E2 -6351.409} C_VEL
LIN {X 0,Y 495.745,Z 55.735,A -85,B 0,C 180,E1 -6354.462,E2 -6354.462} C_VEL
LIN {X 0,Y 495.77,Z 55.725,A -85,B 0,C 180,E1 -6357.406,E2 -6357.406} C_VEL
LIN {X 0,Y 495.767,Z 55.733,A -85,B 0,C 180,E1 -6360.254,E2 -6360.254} C_VEL
LIN {X 0,Y 495.74,Z 55.731,A -85,B 0,C 180,E1 -6360.73,E2 -6360.73} C_VEL
LIN {X 0,Y 495.062,Z 55.814,A -85,B 0,C 180,E1 -6361.409,E2 -6361.409} C_VEL
LIN {X 0,Y 492.182,Z 56.175,A -85,B 0,C 180,E1 -6362.511,E2 -6362.511} C_VEL
LIN {X 0,Y 489.767,Z 56.474,A -85,B 0,C 180,E1 -6363.399,E2 -6363.399} C_VEL
LIN {X 0,Y 488.754,Z 56.607,A -85,B 0,C 180,E1 -6364.085,E2 -6364.085} C_VEL
LIN {X 0,Y 488.685,Z 56.61,A -85,B 0,C 180,E1 -6364.317,E2 -6364.317} C_VEL
LIN {X 0,Y 488.725,Z 56.603,A -85,B 0,C 180,E1 -6367.154,E2 -6367.154} C_VEL
LIN {X 0,Y 488.727,Z 56.61,A -85,B 0,C 180,E1 -6369.811,E2 -6369.811} C_VEL
LIN {X 0,Y 488.705,Z 56.607,A -85,B 0,C 180,E1 -6372.423,E2 -6372.423} C_VEL
LIN {X 0,Y 488.761,Z 56.603,A -85,B 0,C 180,E1 -6375,E2 -6375} C_VEL
LIN {X 0,Y 488.769,Z 56.669,A -85,B 0,C 180,E1 -6377.228,E2 -6377.228} C_VEL
LIN {X 0,Y 489.478,Z 62.114,A -85,B 0,C 180,E1 -6378.404,E2 -6378.404} C_VEL
LIN {X 0,Y 489.426,Z 73.822,A -85,B 0,C 180,E1 -6380.834,E2 -6380.834} C_VEL
LIN {X 0,Y 491.757,Z 86.453,A -85,B 0,C 180,E1 -6381.117,E2 -6381.117} C_VEL
LIN {X 0,Y 491.055,Z 181.139,A -85,B 0,C 180,E1 -6382.522,E2 -6382.522} C_VEL
LIN {X 0,Y 490.872,Z 194.776,A -85,B 0,C 180,E1 -6382.907,E2 -6382.907} C_VEL
LIN {X 0,Y 490.597,Z 207.052,A -85,B 0,C 180,E1 -6383.42,E2 -6383.42} C_VEL
LIN {X 0,Y 490.317,Z 219.577,A -85,B 0,C 180,E1 -6384.139,E2 -6384.139} C_VEL
LIN {X 0,Y 489.896,Z 230.733,A -85,B 0,C 180,E1 -6384.959,E2 -6384.959} C_VEL
LIN {X 0,Y 489.482,Z 240.808,A -85,B 0,C 180,E1 -6385.883,E2 -6385.883} C_VEL
LIN {X 0,Y 489.142,Z 249.872,A -85,B 0,C 180,E1 -6386.912,E2 -6386.912} C_VEL
LIN {X 0,Y 488.741,Z 258.71,A -85,B 0,C 180,E1 -6388.146,E2 -6388.146} C_VEL
LIN {X 0,Y 488.525,Z 265.827,A -85,B 0,C 180,E1 -6389.382,E2 -6389.382} C_VEL
LIN {X 0,Y 488.288,Z 270.65,A -85,B 0,C 180,E1 -6390.413,E2 -6390.413} C_VEL
LIN {X 0,Y 488.061,Z 275.346,A -85,B 0,C 180,E1 -6391.651,E2 -6391.651} C_VEL
LIN {X 0,Y 488.09,Z 278.935,A -85,B 0,C 180,E1 -6392.889,E2 -6392.889} C_VEL
LIN {X 0,Y 487.981,Z 281.542,A -85,B 0,C 180,E1 -6394.13,E2 -6394.13} C_VEL
LIN {X 0,Y 487.928,Z 282.773,A -85,B 0,C 180,E1 -6394.958,E2 -6394.958} C_VEL
LIN {X 0,Y 488.018,Z 283.949,A -85,B 0,C 180,E1 -6396.442,E2 -6396.442} C_VEL
LIN {X 0,Y 487.934,Z 284.002,A -85,B 0,C 180,E1 -6397.449,E2 -6397.449} C_VEL
LIN {X 0,Y 487.933,Z 283.635,A -85,B 0,C 180,E1 -6398.282,E2 -6398.282} C_VEL
LIN {X 0,Y 487.929,Z 282.86,A -85,B 0,C 180,E1 -6399.117,E2 -6399.117} C_VEL
LIN {X 0,Y 488.005,Z 280.026,A -85,B 0,C 180,E1 -6400.791,E2 -6400.791} C_VEL
LIN {X 0,Y 488.147,Z 276.752,A -85,B 0,C 180,E1 -6402.05,E2 -6402.05} C_VEL
LIN {X 0,Y 488.266,Z 272.377,A -85,B 0,C 180,E1 -6403.315,E2 -6403.315} C_VEL
LIN {X 0,Y 488.541,Z 266.77,A -85,B 0,C 180,E1 -6404.581,E2 -6404.581} C_VEL
LIN {X 0,Y 488.785,Z 259.714,A -85,B 0,C 180,E1 -6405.855,E2 -6405.855} C_VEL
LIN {X 0,Y 489.115,Z 250.807,A -85,B 0,C 180,E1 -6407.131,E2 -6407.131} C_VEL
LIN {X 0,Y 489.548,Z 241.633,A -85,B 0,C 180,E1 -6408.195,E2 -6408.195} C_VEL
LIN {X 0,Y 489.94,Z 231.279,A -85,B 0,C 180,E1 -6409.167,E2 -6409.167} C_VEL
LIN {X 0,Y 490.334,Z 219.968,A -85,B 0,C 180,E1 -6410.011,E2 -6410.011} C_VEL
LIN {X 0,Y 490.726,Z 208.047,A -85,B 0,C 180,E1 -6410.706,E2 -6410.706} C_VEL
LIN {X 0,Y 491.08,Z 195.311,A -85,B 0,C 180,E1 -6411.251,E2 -6411.251} C_VEL
LIN {X 0,Y 491.352,Z 182.133,A -85,B 0,C 180,E1 -6411.63,E2 -6411.63} C_VEL
LIN {X 0,Y 491.49,Z 152.366,A -85,B 0,C 180,E1 -6412.102,E2 -6412.102} C_VEL
LIN {X 0,Y 491.936,Z 85.599,A -85,B 0,C 180,E1 -6413.087,E2 -6413.087} C_VEL
LIN {X 0,Y 489.536,Z 73.951,A -85,B 0,C 180,E1 -6413.378,E2 -6413.378} C_VEL
LIN {X 0,Y 489.741,Z 62.761,A -85,B 0,C 180,E1 -6415.728,E2 -6415.728} C_VEL
LIN {X 0,Y 488.753,Z 56.606,A -85,B 0,C 180,E1 -6417.123,E2 -6417.123} C_VEL
LIN {X 0,Y 488.696,Z 56.614,A -85,B 0,C 180,E1 -6420.359,E2 -6420.359} C_VEL
LIN {X 0,Y 488.696,Z 56.611,A -85,B 0,C 180,E1 -6423.476,E2 -6423.476} C_VEL
LIN {X 0,Y 488.648,Z 56.618,A -85,B 0,C 180,E1 -6426.348,E2 -6426.348} C_VEL
LIN {X 0,Y 488.672,Z 56.612,A -85,B 0,C 180,E1 -6429.257,E2 -6429.257} C_VEL
LIN {X 0,Y 488.651,Z 56.614,A -85,B 0,C 180,E1 -6432.53,E2 -6432.53} C_VEL
LIN {X 0,Y 488.699,Z 56.601,A -85,B 0,C 180,E1 -6435.196,E2 -6435.196} C_VEL
LIN {X 0,Y 488.646,Z 56.612,A -85,B 0,C 180,E1 -6438.577,E2 -6438.577} C_VEL
LIN {X 0,Y 488.643,Z 56.618,A -85,B 0,C 180,E1 -6441.796,E2 -6441.796} C_VEL
LIN {X 0,Y 488.708,Z 56.607,A -85,B 0,C 180,E1 -6445.056,E2 -6445.056} C_VEL
LIN {X 0,Y 488.686,Z 56.606,A -85,B 0,C 180,E1 -6448.05,E2 -6448.05} C_VEL
LIN {X 0,Y 488.667,Z 56.615,A -85,B 0,C 180,E1 -6451.319,E2 -6451.319} C_VEL
LIN {X 0,Y 488.67,Z 56.613,A -85,B 0,C 180,E1 -6453.523,E2 -6453.523} C_VEL
LIN {X 0,Y 488.665,Z 56.61,A -85,B 0,C 180,E1 -6456.253,E2 -6456.253} C_VEL
LIN {X 0,Y 488.75,Z 56.605,A -85,B 0,C 180,E1 -6459.176,E2 -6459.176} C_VEL
LIN {X 0,Y 488.751,Z 56.597,A -85,B 0,C 180,E1 -6461.632,E2 -6461.632} C_VEL
LIN {X 0,Y 488.755,Z 56.604,A -85,B 0,C 180,E1 -6464.999,E2 -6464.999} C_VEL
LIN {X 0,Y 488.807,Z 56.593,A -85,B 0,C 180,E1 -6468.387,E2 -6468.387} C_VEL
LIN {X 0,Y 488.766,Z 56.599,A -85,B 0,C 180,E1 -6471.733,E2 -6471.733} C_VEL
LIN {X 0,Y 488.807,Z 56.593,A -85,B 0,C 180,E1 -6474.223,E2 -6474.223} C_VEL
LIN {X 0,Y 488.952,Z 56.576,A -85,B 0,C 180,E1 -6477.528,E2 -6477.528} C_VEL
LIN {X 0,Y 488.896,Z 56.581,A -85,B 0,C 180,E1 -6480.823,E2 -6480.823} C_VEL
LIN {X 0,Y 488.945,Z 56.579,A -85,B 0,C 180,E1 -6482.471,E2 -6482.471} C_VEL
LIN {X 0,Y 488.818,Z 56.593,A -85,B 0,C 180,E1 -6485.776,E2 -6485.776} C_VEL
LIN {X 0,Y 488.766,Z 56.601,A -85,B 0,C 180,E1 -6488.267,E2 -6488.267} C_VEL
LIN {X 0,Y 488.809,Z 56.594,A -85,B 0,C 180,E1 -6491.612,E2 -6491.612} C_VEL
LIN {X 0,Y 488.758,Z 56.6,A -85,B 0,C 180,E1 -6495,E2 -6495} C_VEL
LIN {X 0,Y 488.747,Z 56.599,A -85,B 0,C 180,E1 -6498.442,E2 -6498.442} C_VEL
LIN {X 0,Y 488.71,Z 56.608,A -85,B 0,C 180,E1 -6501.071,E2 -6501.071} C_VEL
LIN {X 0,Y 488.673,Z 56.613,A -85,B 0,C 180,E1 -6503.746,E2 -6503.746} C_VEL
LIN {X 0,Y 488.75,Z 56.603,A -85,B 0,C 180,E1 -6506.933,E2 -6506.933} C_VEL
LIN {X 0,Y 488.724,Z 56.609,A -85,B 0,C 180,E1 -6509.27,E2 -6509.27} C_VEL
LIN {X 0,Y 488.705,Z 56.605,A -85,B 0,C 180,E1 -6512.147,E2 -6512.147} C_VEL
LIN {X 0,Y 488.721,Z 56.601,A -85,B 0,C 180,E1 -6515.115,E2 -6515.115} C_VEL
LIN {X 0,Y 488.682,Z 56.606,A -85,B 0,C 180,E1 -6518.2,E2 -6518.2} C_VEL
LIN {X 0,Y 488.721,Z 56.607,A -85,B 0,C 180,E1 -6520.344,E2 -6520.344} C_VEL
LIN {X 0,Y 488.687,Z 56.608,A -85,B 0,C 180,E1 -6523.655,E2 -6523.655} C_VEL
LIN {X 0,Y 488.687,Z 56.612,A -85,B 0,C 180,E1 -6526.345,E2 -6526.345} C_VEL
LIN {X 0,Y 488.736,Z 56.602,A -85,B 0,C 180,E1 -6529.676,E2 -6529.676} C_VEL
LIN {X 0,Y 488.682,Z 56.611,A -85,B 0,C 180,E1 -6532.841,E2 -6532.841} C_VEL
LIN {X 0,Y 488.733,Z 56.607,A -85,B 0,C 180,E1 -6535.887,E2 -6535.887} C_VEL
LIN {X 0,Y 488.695,Z 56.612,A -85,B 0,C 180,E1 -6538.82,E2 -6538.82} C_VEL
LIN {X 0,Y 488.746,Z 56.608,A -85,B 0,C 180,E1 -6541.671,E2 -6541.671} C_VEL
LIN {X 0,Y 488.787,Z 56.729,A -85,B 0,C 180,E1 -6544.017,E2 -6544.017} C_VEL
LIN {X 0,Y 490.803,Z 67.265,A -85,B 0,C 180,E1 -6545.914,E2 -6545.914} C_VEL
LIN {X 0,Y 490.396,Z 79.259,A -85,B 0,C 180,E1 -6547.901,E2 -6547.901} C_VEL
LIN {X 0,Y 489.751,Z 97.697,A -85,B 0,C 180,E1 -6550.909,E2 -6550.909} C_VEL
LIN {X 0,Y 489.222,Z 114.823,A -85,B 0,C 180,E1 -6553.664,E2 -6553.664} C_VEL
LIN {X 0,Y 491.713,Z 132.52,A -85,B 0,C 180,E1 -6554.024,E2 -6554.024} C_VEL
LIN {X 0,Y 491.139,Z 223.84,A -85,B 0,C 180,E1 -6555.392,E2 -6555.392} C_VEL
LIN {X 0,Y 490.801,Z 237.721,A -85,B 0,C 180,E1 -6555.778,E2 -6555.778} C_VEL
LIN {X 0,Y 490.416,Z 249.613,A -85,B 0,C 180,E1 -6556.269,E2 -6556.269} C_VEL
LIN {X 0,Y 489.979,Z 261.986,A -85,B 0,C 180,E1 -6556.964,E2 -6556.964} C_VEL
LIN {X 0,Y 489.471,Z 273.178,A -85,B 0,C 180,E1 -6557.773,E2 -6557.773} C_VEL
LIN {X 0,Y 489.097,Z 283.565,A -85,B 0,C 180,E1 -6558.709,E2 -6558.709} C_VEL
LIN {X 0,Y 488.74,Z 292.069,A -85,B 0,C 180,E1 -6559.645,E2 -6559.645} C_VEL
LIN {X 0,Y 488.42,Z 301.302,A -85,B 0,C 180,E1 -6560.893,E2 -6560.893} C_VEL
LIN {X 0,Y 488.192,Z 308.737,A -85,B 0,C 180,E1 -6562.139,E2 -6562.139} C_VEL
LIN {X 0,Y 487.999,Z 315.527,A -85,B 0,C 180,E1 -6563.574,E2 -6563.574} C_VEL
LIN {X 0,Y 487.962,Z 320.754,A -85,B 0,C 180,E1 -6565.042,E2 -6565.042} C_VEL
LIN {X 0,Y 487.929,Z 323.056,A -85,B 0,C 180,E1 -6565.87,E2 -6565.87} C_VEL
LIN {X 0,Y 487.977,Z 324.923,A -85,B 0,C 180,E1 -6566.697,E2 -6566.697} C_VEL
LIN {X 0,Y 487.937,Z 326.32,A -85,B 0,C 180,E1 -6567.523,E2 -6567.523} C_VEL
LIN {X 0,Y 487.895,Z 327.317,A -85,B 0,C 180,E1 -6568.349,E2 -6568.349} C_VEL
LIN {X 0,Y 487.838,Z 328.139,A -85,B 0,C 180,E1 -6570,E2 -6570} C_VEL
LIN {X 0,Y 487.895,Z 327.311,A -85,B 0,C 180,E1 -6571.651,E2 -6571.651} C_VEL
LIN {X 0,Y 487.937,Z 326.311,A -85,B 0,C 180,E1 -6572.476,E2 -6572.476} C_VEL
LIN {X 0,Y 487.977,Z 324.906,A -85,B 0,C 180,E1 -6573.302,E2 -6573.302} C_VEL
LIN {X 0,Y 487.918,Z 321.947,A -85,B 0,C 180,E1 -6574.544,E2 -6574.544} C_VEL
LIN {X 0,Y 487.976,Z 317.946,A -85,B 0,C 180,E1 -6575.786,E2 -6575.786} C_VEL
LIN {X 0,Y 488.129,Z 311.788,A -85,B 0,C 180,E1 -6577.237,E2 -6577.237} C_VEL
LIN {X 0,Y 488.296,Z 305.058,A -85,B 0,C 180,E1 -6578.483,E2 -6578.483} C_VEL
LIN {X 0,Y 488.551,Z 296.707,A -85,B 0,C 180,E1 -6579.731,E2 -6579.731} C_VEL
LIN {X 0,Y 488.893,Z 288.13,A -85,B 0,C 180,E1 -6580.77,E2 -6580.77} C_VEL
LIN {X 0,Y 489.314,Z 277.536,A -85,B 0,C 180,E1 -6581.81,E2 -6581.81} C_VEL
LIN {X 0,Y 489.703,Z 266.106,A -85,B 0,C 180,E1 -6582.71,E2 -6582.71} C_VEL
LIN {X 0,Y 490.089,Z 255.493,A -85,B 0,C 180,E1 -6583.37,E2 -6583.37} C_VEL
LIN {X 0,Y 490.481,Z 243.52,A -85,B 0,C 180,E1 -6583.94,E2 -6583.94} C_VEL
LIN {X 0,Y 490.87,Z 230.588,A -85,B 0,C 180,E1 -6584.378,E2 -6584.378} C_VEL
LIN {X 0,Y 491.086,Z 216.911,A -85,B 0,C 180,E1 -6584.662,E2 -6584.662} C_VEL
LIN {X 0,Y 491.518,Z 131.516,A -85,B 0,C 180,E1 -6585.911,E2 -6585.911} C_VEL
LIN {X 0,Y 489.159,Z 114.984,A -85,B 0,C 180,E1 -6586.228,E2 -6586.228} C_VEL
LIN {X 0,Y 489.751,Z 94.476,A -85,B 0,C 180,E1 -6589.49,E2 -6589.49} C_VEL
LIN {X 0,Y 490.478,Z 72.878,A -85,B 0,C 180,E1 -6592.964,E2 -6592.964} C_VEL
LIN {X 0,Y 490.552,Z 65.945,A -85,B 0,C 180,E1 -6594.099,E2 -6594.099} C_VEL
LIN {X 0,Y 488.797,Z 56.601,A -85,B 0,C 180,E1 -6595.724,E2 -6595.724} C_VEL
LIN {X 0,Y 488.732,Z 56.606,A -85,B 0,C 180,E1 -6598.695,E2 -6598.695} C_VEL
LIN {X 0,Y 488.693,Z 56.607,A -85,B 0,C 180,E1 -6601.179,E2 -6601.179} C_VEL
LIN {X 0,Y 488.731,Z 56.607,A -85,B 0,C 180,E1 -6604.113,E2 -6604.113} C_VEL
LIN {X 0,Y 488.68,Z 56.61,A -85,B 0,C 180,E1 -6607.159,E2 -6607.159} C_VEL
LIN {X 0,Y 488.718,Z 56.604,A -85,B 0,C 180,E1 -6610.344,E2 -6610.344} C_VEL
LIN {X 0,Y 488.684,Z 56.615,A -85,B 0,C 180,E1 -6613.654,E2 -6613.654} C_VEL
LIN {X 0,Y 488.684,Z 56.608,A -85,B 0,C 180,E1 -6616.345,E2 -6616.345} C_VEL
LIN {X 0,Y 488.733,Z 56.606,A -85,B 0,C 180,E1 -6619.676,E2 -6619.676} C_VEL
LIN {X 0,Y 488.679,Z 56.611,A -85,B 0,C 180,E1 -6622.841,E2 -6622.841} C_VEL
LIN {X 0,Y 488.732,Z 56.602,A -85,B 0,C 180,E1 -6625.887,E2 -6625.887} C_VEL
LIN {X 0,Y 488.692,Z 56.612,A -85,B 0,C 180,E1 -6628.82,E2 -6628.82} C_VEL
LIN {X 0,Y 488.743,Z 56.601,A -85,B 0,C 180,E1 -6631.671,E2 -6631.671} C_VEL
LIN {X 0,Y 488.745,Z 56.603,A -85,B 0,C 180,E1 -6634.444,E2 -6634.444} C_VEL
LIN {X 0,Y 488.721,Z 56.607,A -85,B 0,C 180,E1 -6637.153,E2 -6637.153} C_VEL
LIN {X 0,Y 488.724,Z 56.603,A -85,B 0,C 180,E1 -6639.811,E2 -6639.811} C_VEL
LIN {X 0,Y 488.714,Z 56.609,A -85,B 0,C 180,E1 -6642.423,E2 -6642.423} C_VEL
LIN {X 0,Y 488.761,Z 56.601,A -85,B 0,C 180,E1 -6645,E2 -6645} C_VEL
LIN {X 0,Y 488.805,Z 56.6,A -85,B 0,C 180,E1 -6648.388,E2 -6648.388} C_VEL
LIN {X 0,Y 488.815,Z 56.593,A -85,B 0,C 180,E1 -6651.734,E2 -6651.734} C_VEL
LIN {X 0,Y 488.848,Z 56.595,A -85,B 0,C 180,E1 -6654.224,E2 -6654.224} C_VEL
LIN {X 0,Y 488.955,Z 56.575,A -85,B 0,C 180,E1 -6657.529,E2 -6657.529} C_VEL
LIN {X 0,Y 488.914,Z 56.58,A -85,B 0,C 180,E1 -6660.824,E2 -6660.824} C_VEL
LIN {X 0,Y 488.955,Z 56.577,A -85,B 0,C 180,E1 -6662.472,E2 -6662.472} C_VEL
LIN {X 0,Y 488.838,Z 56.595,A -85,B 0,C 180,E1 -6665.776,E2 -6665.776} C_VEL
LIN {X 0,Y 488.785,Z 56.598,A -85,B 0,C 180,E1 -6668.267,E2 -6668.267} C_VEL
LIN {X 0,Y 488.806,Z 56.599,A -85,B 0,C 180,E1 -6671.613,E2 -6671.613} C_VEL
LIN {X 0,Y 488.76,Z 56.6,A -85,B 0,C 180,E1 -6675.001,E2 -6675.001} C_VEL
LIN {X 0,Y 488.746,Z 56.6,A -85,B 0,C 180,E1 -6678.443,E2 -6678.443} C_VEL
LIN {X 0,Y 488.707,Z 56.609,A -85,B 0,C 180,E1 -6681.071,E2 -6681.071} C_VEL
LIN {X 0,Y 488.671,Z 56.612,A -85,B 0,C 180,E1 -6683.747,E2 -6683.747} C_VEL
LIN {X 0,Y 488.748,Z 56.604,A -85,B 0,C 180,E1 -6686.934,E2 -6686.934} C_VEL
LIN {X 0,Y 488.722,Z 56.61,A -85,B 0,C 180,E1 -6689.271,E2 -6689.271} C_VEL
LIN {X 0,Y 488.703,Z 56.605,A -85,B 0,C 180,E1 -6692.147,E2 -6692.147} C_VEL
LIN {X 0,Y 488.715,Z 56.61,A -85,B 0,C 180,E1 -6695.116,E2 -6695.116} C_VEL
LIN {X 0,Y 488.678,Z 56.609,A -85,B 0,C 180,E1 -6698.201,E2 -6698.201} C_VEL
LIN {X 0,Y 488.694,Z 56.609,A -85,B 0,C 180,E1 -6700.341,E2 -6700.341} C_VEL
LIN {X 0,Y 488.676,Z 56.609,A -85,B 0,C 180,E1 -6703.656,E2 -6703.656} C_VEL
LIN {X 0,Y 488.68,Z 56.613,A -85,B 0,C 180,E1 -6706.345,E2 -6706.345} C_VEL
LIN {X 0,Y 488.705,Z 56.605,A -85,B 0,C 180,E1 -6709.674,E2 -6709.674} C_VEL
LIN {X 0,Y 488.669,Z 56.613,A -85,B 0,C 180,E1 -6712.84,E2 -6712.84} C_VEL
LIN {X 0,Y 488.729,Z 56.605,A -85,B 0,C 180,E1 -6715.887,E2 -6715.887} C_VEL
LIN {X 0,Y 488.695,Z 56.608,A -85,B 0,C 180,E1 -6718.821,E2 -6718.821} C_VEL
LIN {X 0,Y 488.713,Z 56.607,A -85,B 0,C 180,E1 -6721.669,E2 -6721.669} C_VEL
LIN {X 0,Y 488.685,Z 56.61,A -85,B 0,C 180,E1 -6724.317,E2 -6724.317} C_VEL
LIN {X 0,Y 488.053,Z 56.693,A -85,B 0,C 180,E1 -6725.005,E2 -6725.005} C_VEL
LIN {X 0,Y 485.211,Z 57.051,A -85,B 0,C 180,E1 -6726.122,E2 -6726.122} C_VEL
LIN {X 0,Y 482.781,Z 57.351,A -85,B 0,C 180,E1 -6727.023,E2 -6727.023} C_VEL
LIN {X 0,Y 481.728,Z 57.479,A -85,B 0,C 180,E1 -6727.718,E2 -6727.718} C_VEL
LIN {X 0,Y 481.639,Z 57.488,A -85,B 0,C 180,E1 -6727.954,E2 -6727.954} C_VEL
LIN {X 0,Y 481.704,Z 57.479,A -85,B 0,C 180,E1 -6730.393,E2 -6730.393} C_VEL
LIN {X 0,Y 481.671,Z 57.482,A -85,B 0,C 180,E1 -6733.033,E2 -6733.033} C_VEL
LIN {X 0,Y 481.686,Z 57.488,A -85,B 0,C 180,E1 -6735.639,E2 -6735.639} C_VEL
LIN {X 0,Y 481.725,Z 57.531,A -85,B 0,C 180,E1 -6737.092,E2 -6737.092} C_VEL
LIN {X 0,Y 482.53,Z 63.762,A -85,B 0,C 180,E1 -6738.448,E2 -6738.448} C_VEL
LIN {X 0,Y 482.483,Z 74.134,A -85,B 0,C 180,E1 -6740.622,E2 -6740.622} C_VEL
LIN {X 0,Y 484.909,Z 87.115,A -85,B 0,C 180,E1 -6740.911,E2 -6740.911} C_VEL
LIN {X 0,Y 484.186,Z 180.578,A -85,B 0,C 180,E1 -6742.31,E2 -6742.31} C_VEL
LIN {X 0,Y 484.01,Z 193.763,A -85,B 0,C 180,E1 -6742.675,E2 -6742.675} C_VEL
LIN {X 0,Y 483.668,Z 206.969,A -85,B 0,C 180,E1 -6743.22,E2 -6743.22} C_VEL
LIN {X 0,Y 483.472,Z 218.038,A -85,B 0,C 180,E1 -6743.846,E2 -6743.846} C_VEL
LIN {X 0,Y 482.968,Z 229.551,A -85,B 0,C 180,E1 -6744.677,E2 -6744.677} C_VEL
LIN {X 0,Y 482.536,Z 239.9,A -85,B 0,C 180,E1 -6745.615,E2 -6745.615} C_VEL
LIN {X 0,Y 482.186,Z 249.236,A -85,B 0,C 180,E1 -6746.658,E2 -6746.658} C_VEL
LIN {X 0,Y 481.762,Z 258.244,A -85,B 0,C 180,E1 -6747.91,E2 -6747.91} C_VEL
LIN {X 0,Y 481.487,Z 265.506,A -85,B 0,C 180,E1 -6749.164,E2 -6749.164} C_VEL
LIN {X 0,Y 481.204,Z 271.346,A -85,B 0,C 180,E1 -6750.419,E2 -6750.419} C_VEL
LIN {X 0,Y 480.984,Z 275.962,A -85,B 0,C 180,E1 -6751.675,E2 -6751.675} C_VEL
LIN {X 0,Y 481.003,Z 278.424,A -85,B 0,C 180,E1 -6752.513,E2 -6752.513} C_VEL
LIN {X 0,Y 480.973,Z 280.421,A -85,B 0,C 180,E1 -6753.351,E2 -6753.351} C_VEL
LIN {X 0,Y 480.856,Z 283.207,A -85,B 0,C 180,E1 -6755.031,E2 -6755.031} C_VEL
LIN {X 0,Y 480.934,Z 284.264,A -85,B 0,C 180,E1 -6756.431,E2 -6756.431} C_VEL
LIN {X 0,Y 480.846,Z 284.307,A -85,B 0,C 180,E1 -6757.559,E2 -6757.559} C_VEL
LIN {X 0,Y 480.837,Z 283.904,A -85,B 0,C 180,E1 -6758.405,E2 -6758.405} C_VEL
LIN {X 0,Y 480.835,Z 283.063,A -85,B 0,C 180,E1 -6759.252,E2 -6759.252} C_VEL
LIN {X 0,Y 480.875,Z 281.814,A -85,B 0,C 180,E1 -6760.101,E2 -6760.101} C_VEL
LIN {X 0,Y 481.004,Z 279.173,A -85,B 0,C 180,E1 -6761.367,E2 -6761.367} C_VEL
LIN {X 0,Y 481.134,Z 275.446,A -85,B 0,C 180,E1 -6762.657,E2 -6762.657} C_VEL
LIN {X 0,Y 481.298,Z 270.591,A -85,B 0,C 180,E1 -6763.942,E2 -6763.942} C_VEL
LIN {X 0,Y 481.549,Z 264.428,A -85,B 0,C 180,E1 -6765.231,E2 -6765.231} C_VEL
LIN {X 0,Y 481.908,Z 256.712,A -85,B 0,C 180,E1 -6766.522,E2 -6766.522} C_VEL
LIN {X 0,Y 482.277,Z 248.746,A -85,B 0,C 180,E1 -6767.601,E2 -6767.601} C_VEL
LIN {X 0,Y 482.727,Z 238.966,A -85,B 0,C 180,E1 -6768.681,E2 -6768.681} C_VEL
LIN {X 0,Y 483.174,Z 228.038,A -85,B 0,C 180,E1 -6769.656,E2 -6769.656} C_VEL
LIN {X 0,Y 483.613,Z 217.325,A -85,B 0,C 180,E1 -6770.413,E2 -6770.413} C_VEL
LIN {X 0,Y 483.99,Z 205.467,A -85,B 0,C 180,E1 -6771.063,E2 -6771.063} C_VEL
LIN {X 0,Y 484.326,Z 192.027,A -85,B 0,C 180,E1 -6771.601,E2 -6771.601} C_VEL
LIN {X 0,Y 484.558,Z 179.376,A -85,B 0,C 180,E1 -6771.926,E2 -6771.926} C_VEL
LIN {X 0,Y 485.186,Z 86.583,A -85,B 0,C 180,E1 -6773.328,E2 -6773.328} C_VEL
LIN {X 0,Y 482.624,Z 74.324,A -85,B 0,C 180,E1 -6773.626,E2 -6773.626} C_VEL
LIN {X 0,Y 482.74,Z 63.658,A -85,B 0,C 180,E1 -6775.897,E2 -6775.897} C_VEL
LIN {X 0,Y 481.703,Z 57.484,A -85,B 0,C 180,E1 -6777.293,E2 -6777.293} C_VEL
LIN {X 0,Y 481.633,Z 57.492,A -85,B 0,C 180,E1 -6780.712,E2 -6780.712} C_VEL
LIN {X 0,Y 481.653,Z 57.49,A -85,B 0,C 180,E1 -6783.724,E2 -6783.724} C_VEL
LIN {X 0,Y 481.607,Z 57.491,A -85,B 0,C 180,E1 -6786.749,E2 -6786.749} C_VEL
LIN {X 0,Y 481.632,Z 57.494,A -85,B 0,C 180,E1 -6789.945,E2 -6789.945} C_VEL
LIN {X 0,Y 481.617,Z 57.491,A -85,B 0,C 180,E1 -6793.303,E2 -6793.303} C_VEL
LIN {X 0,Y 481.651,Z 57.484,A -85,B 0,C 180,E1 -6795.642,E2 -6795.642} C_VEL
LIN {X 0,Y 481.607,Z 57.489,A -85,B 0,C 180,E1 -6798.953,E2 -6798.953} C_VEL
LIN {X 0,Y 481.619,Z 57.491,A -85,B 0,C 180,E1 -6801.999,E2 -6801.999} C_VEL
LIN {X 0,Y 481.673,Z 57.486,A -85,B 0,C 180,E1 -6805.316,E2 -6805.316} C_VEL
LIN {X 0,Y 481.623,Z 57.485,A -85,B 0,C 180,E1 -6808.31,E2 -6808.31} C_VEL
LIN {X 0,Y 481.639,Z 57.492,A -85,B 0,C 180,E1 -6811.214,E2 -6811.214} C_VEL
LIN {X 0,Y 481.62,Z 57.488,A -85,B 0,C 180,E1 -6814.038,E2 -6814.038} C_VEL
LIN {X 0,Y 481.657,Z 57.488,A -85,B 0,C 180,E1 -6816.818,E2 -6816.818} C_VEL
LIN {X 0,Y 481.697,Z 57.48,A -85,B 0,C 180,E1 -6819.502,E2 -6819.502} C_VEL
LIN {X 0,Y 481.689,Z 57.477,A -85,B 0,C 180,E1 -6822.157,E2 -6822.157} C_VEL
LIN {X 0,Y 481.74,Z 57.481,A -85,B 0,C 180,E1 -6824.775,E2 -6824.775} C_VEL
LIN {X 0,Y 481.753,Z 57.47,A -85,B 0,C 180,E1 -6828.215,E2 -6828.215} C_VEL
LIN {X 0,Y 481.724,Z 57.475,A -85,B 0,C 180,E1 -6831.611,E2 -6831.611} C_VEL
LIN {X 0,Y 481.768,Z 57.469,A -85,B 0,C 180,E1 -6834.139,E2 -6834.139} C_VEL
LIN {X 0,Y 481.919,Z 57.452,A -85,B 0,C 180,E1 -6837.492,E2 -6837.492} C_VEL
LIN {X 0,Y 481.913,Z 57.452,A -85,B 0,C 180,E1 -6840,E2 -6840} C_VEL
LIN {X 0,Y 481.911,Z 57.455,A -85,B 0,C 180,E1 -6842.507,E2 -6842.507} C_VEL
LIN {X 0,Y 481.779,Z 57.469,A -85,B 0,C 180,E1 -6845.861,E2 -6845.861} C_VEL
LIN {X 0,Y 481.725,Z 57.477,A -85,B 0,C 180,E1 -6848.389,E2 -6848.389} C_VEL
LIN {X 0,Y 481.754,Z 57.472,A -85,B 0,C 180,E1 -6851.785,E2 -6851.785} C_VEL
LIN {X 0,Y 481.742,Z 57.476,A -85,B 0,C 180,E1 -6855.224,E2 -6855.224} C_VEL
LIN {X 0,Y 481.709,Z 57.476,A -85,B 0,C 180,E1 -6858.722,E2 -6858.722} C_VEL
LIN {X 0,Y 481.648,Z 57.488,A -85,B 0,C 180,E1 -6861.395,E2 -6861.395} C_VEL
LIN {X 0,Y 481.652,Z 57.485,A -85,B 0,C 180,E1 -6864.114,E2 -6864.114} C_VEL
LIN {X 0,Y 481.717,Z 57.479,A -85,B 0,C 180,E1 -6867.131,E2 -6867.131} C_VEL
LIN {X 0,Y 481.68,Z 57.481,A -85,B 0,C 180,E1 -6869.741,E2 -6869.741} C_VEL
LIN {X 0,Y 481.675,Z 57.485,A -85,B 0,C 180,E1 -6872.674,E2 -6872.674} C_VEL
LIN {X 0,Y 481.64,Z 57.478,A -85,B 0,C 180,E1 -6875.709,E2 -6875.709} C_VEL
LIN {X 0,Y 481.673,Z 57.488,A -85,B 0,C 180,E1 -6878.859,E2 -6878.859} C_VEL
LIN {X 0,Y 481.655,Z 57.484,A -85,B 0,C 180,E1 -6881.913,E2 -6881.913} C_VEL
LIN {X 0,Y 481.657,Z 57.49,A -85,B 0,C 180,E1 -6884.458,E2 -6884.458} C_VEL
LIN {X 0,Y 481.65,Z 57.485,A -85,B 0,C 180,E1 -6887.839,E2 -6887.839} C_VEL
LIN {X 0,Y 481.683,Z 57.485,A -85,B 0,C 180,E1 -6890.651,E2 -6890.651} C_VEL
LIN {X 0,Y 481.63,Z 57.488,A -85,B 0,C 180,E1 -6893.376,E2 -6893.376} C_VEL
LIN {X 0,Y 481.713,Z 57.485,A -85,B 0,C 180,E1 -6896.33,E2 -6896.33} C_VEL
LIN {X 0,Y 481.653,Z 57.49,A -85,B 0,C 180,E1 -6899.417,E2 -6899.417} C_VEL
LIN {X 0,Y 481.702,Z 57.485,A -85,B 0,C 180,E1 -6902.168,E2 -6902.168} C_VEL
LIN {X 0,Y 481.759,Z 57.615,A -85,B 0,C 180,E1 -6903.784,E2 -6903.784} C_VEL
LIN {X 0,Y 483.858,Z 68.464,A -85,B 0,C 180,E1 -6905.774,E2 -6905.774} C_VEL
LIN {X 0,Y 483.553,Z 79.112,A -85,B 0,C 180,E1 -6907.572,E2 -6907.572} C_VEL
LIN {X 0,Y 482.813,Z 97.697,A -85,B 0,C 180,E1 -6910.652,E2 -6910.652} C_VEL
LIN {X 0,Y 482.283,Z 114.788,A -85,B 0,C 180,E1 -6913.409,E2 -6913.409} C_VEL
LIN {X 0,Y 484.942,Z 133.269,A -85,B 0,C 180,E1 -6913.791,E2 -6913.791} C_VEL
LIN {X 0,Y 484.347,Z 223.185,A -85,B 0,C 180,E1 -6915.155,E2 -6915.155} C_VEL
LIN {X 0,Y 483.951,Z 236.408,A -85,B 0,C 180,E1 -6915.519,E2 -6915.519} C_VEL
LIN {X 0,Y 483.535,Z 248.549,A -85,B 0,C 180,E1 -6916.016,E2 -6916.016} C_VEL
LIN {X 0,Y 483.114,Z 260.171,A -85,B 0,C 180,E1 -6916.658,E2 -6916.658} C_VEL
LIN {X 0,Y 482.567,Z 272.138,A -85,B 0,C 180,E1 -6917.518,E2 -6917.518} C_VEL
LIN {X 0,Y 482.179,Z 282.339,A -85,B 0,C 180,E1 -6918.439,E2 -6918.439} C_VEL
LIN {X 0,Y 481.712,Z 291.878,A -85,B 0,C 180,E1 -6919.492,E2 -6919.492} C_VEL
LIN {X 0,Y 481.369,Z 301.075,A -85,B 0,C 180,E1 -6920.758,E2 -6920.758} C_VEL
LIN {X 0,Y 481.14,Z 308.491,A -85,B 0,C 180,E1 -6922.023,E2 -6922.023} C_VEL
LIN {X 0,Y 480.959,Z 314.451,A -85,B 0,C 180,E1 -6923.287,E2 -6923.287} C_VEL
LIN {X 0,Y 480.908,Z 319.165,A -85,B 0,C 180,E1 -6924.549,E2 -6924.549} C_VEL
LIN {X 0,Y 480.828,Z 322.765,A -85,B 0,C 180,E1 -6925.809,E2 -6925.809} C_VEL
LIN {X 0,Y 480.9,Z 324.624,A -85,B 0,C 180,E1 -6926.648,E2 -6926.648} C_VEL
LIN {X 0,Y 480.826,Z 327.009,A -85,B 0,C 180,E1 -6928.325,E2 -6928.325} C_VEL
LIN {X 0,Y 480.772,Z 327.612,A -85,B 0,C 180,E1 -6929.162,E2 -6929.162} C_VEL
LIN {X 0,Y 480.761,Z 327.819,A -85,B 0,C 180,E1 -6930,E2 -6930} C_VEL
LIN {X 0,Y 480.826,Z 326.98,A -85,B 0,C 180,E1 -6931.675,E2 -6931.675} C_VEL
LIN {X 0,Y 480.849,Z 325.975,A -85,B 0,C 180,E1 -6932.513,E2 -6932.513} C_VEL
LIN {X 0,Y 480.9,Z 324.562,A -85,B 0,C 180,E1 -6933.351,E2 -6933.351} C_VEL
LIN {X 0,Y 480.836,Z 321.594,A -85,B 0,C 180,E1 -6934.611,E2 -6934.611} C_VEL
LIN {X 0,Y 480.864,Z 316.676,A -85,B 0,C 180,E1 -6936.109,E2 -6936.109} C_VEL
LIN {X 0,Y 481.073,Z 310.382,A -85,B 0,C 180,E1 -6937.555,E2 -6937.555} C_VEL
LIN {X 0,Y 481.252,Z 303.404,A -85,B 0,C 180,E1 -6938.82,E2 -6938.82} C_VEL
LIN {X 0,Y 481.541,Z 294.655,A -85,B 0,C 180,E1 -6940.086,E2 -6940.086} C_VEL
LIN {X 0,Y 481.959,Z 285.697,A -85,B 0,C 180,E1 -6941.14,E2 -6941.14} C_VEL
LIN {X 0,Y 482.36,Z 275.076,A -85,B 0,C 180,E1 -6942.159,E2 -6942.159} C_VEL
LIN {X 0,Y 482.857,Z 263.44,A -85,B 0,C 180,E1 -6943.038,E2 -6943.038} C_VEL
LIN {X 0,Y 483.224,Z 252.857,A -85,B 0,C 180,E1 -6943.67,E2 -6943.67} C_VEL
LIN {X 0,Y 483.66,Z 240.151,A -85,B 0,C 180,E1 -6944.248,E2 -6944.248} C_VEL
LIN {X 0,Y 484.006,Z 227.684,A -85,B 0,C 180,E1 -6944.64,E2 -6944.64} C_VEL
LIN {X 0,Y 484.209,Z 211.773,A -85,B 0,C 180,E1 -6944.929,E2 -6944.929} C_VEL
LIN {X 0,Y 484.618,Z 131.981,A -85,B 0,C 180,E1 -6946.113,E2 -6946.113} C_VEL
LIN {X 0,Y 482.152,Z 114.655,A -85,B 0,C 180,E1 -6946.452,E2 -6946.452} C_VEL
LIN {X 0,Y 482.759,Z 95.376,A -85,B 0,C 180,E1 -6949.562,E2 -6949.562} C_VEL
LIN {X 0,Y 483.463,Z 75.017,A -85,B 0,C 180,E1 -6952.883,E2 -6952.883} C_VEL
LIN {X 0,Y 483.652,Z 68.211,A -85,B 0,C 180,E1 -6954.008,E2 -6954.008} C_VEL
LIN {X 0,Y 481.748,Z 57.48,A -85,B 0,C 180,E1 -6955.912,E2 -6955.912} C_VEL
LIN {X 0,Y 481.679,Z 57.484,A -85,B 0,C 180,E1 -6958.903,E2 -6958.903} C_VEL
LIN {X 0,Y 481.658,Z 57.488,A -85,B 0,C 180,E1 -6962.189,E2 -6962.189} C_VEL
LIN {X 0,Y 481.689,Z 57.479,A -85,B 0,C 180,E1 -6964.682,E2 -6964.682} C_VEL
LIN {X 0,Y 481.656,Z 57.488,A -85,B 0,C 180,E1 -6968.007,E2 -6968.007} C_VEL
LIN {X 0,Y 481.656,Z 57.485,A -85,B 0,C 180,E1 -6971.042,E2 -6971.042} C_VEL
LIN {X 0,Y 481.654,Z 57.484,A -85,B 0,C 180,E1 -6974.458,E2 -6974.458} C_VEL
LIN {X 0,Y 481.647,Z 57.487,A -85,B 0,C 180,E1 -6977.839,E2 -6977.839} C_VEL
LIN {X 0,Y 481.66,Z 57.484,A -85,B 0,C 180,E1 -6980.654,E2 -6980.654} C_VEL
LIN {X 0,Y 481.627,Z 57.493,A -85,B 0,C 180,E1 -6983.376,E2 -6983.376} C_VEL
LIN {X 0,Y 481.709,Z 57.477,A -85,B 0,C 180,E1 -6986.33,E2 -6986.33} C_VEL
LIN {X 0,Y 481.65,Z 57.487,A -85,B 0,C 180,E1 -6989.417,E2 -6989.417} C_VEL
LIN {X 0,Y 481.699,Z 57.478,A -85,B 0,C 180,E1 -6992.168,E2 -6992.168} C_VEL
LIN {X 0,Y 481.715,Z 57.483,A -85,B 0,C 180,E1 -6994.97,E2 -6994.97} C_VEL
LIN {X 0,Y 481.648,Z 57.484,A -85,B 0,C 180,E1 -6997.705,E2 -6997.705} C_VEL
LIN {X 0,Y 481.704,Z 57.481,A -85,B 0,C 180,E1 -7000.393,E2 -7000.393} C_VEL
LIN {X 0,Y 481.678,Z 57.484,A -85,B 0,C 180,E1 -7003.034,E2 -7003.034} C_VEL
LIN {X 0,Y 481.687,Z 57.479,A -85,B 0,C 180,E1 -7005.639,E2 -7005.639} C_VEL
LIN {X 0,Y 481.75,Z 57.476,A -85,B 0,C 180,E1 -7008.215,E2 -7008.215} C_VEL
LIN {X 0,Y 481.761,Z 57.471,A -85,B 0,C 180,E1 -7011.612,E2 -7011.612} C_VEL
LIN {X 0,Y 481.809,Z 57.471,A -85,B 0,C 180,E1 -7014.14,E2 -7014.14} C_VEL
LIN {X 0,Y 481.921,Z 57.451,A -85,B 0,C 180,E1 -7017.493,E2 -7017.493} C_VEL
LIN {X 0,Y 481.941,Z 57.455,A -85,B 0,C 180,E1 -7020,E2 -7020} C_VEL
LIN {X 0,Y 481.921,Z 57.452,A -85,B 0,C 180,E1 -7022.508,E2 -7022.508} C_VEL
LIN {X 0,Y 481.797,Z 57.473,A -85,B 0,C 180,E1 -7025.861,E2 -7025.861} C_VEL
LIN {X 0,Y 481.74,Z 57.474,A -85,B 0,C 180,E1 -7028.389,E2 -7028.389} C_VEL
LIN {X 0,Y 481.751,Z 57.479,A -85,B 0,C 180,E1 -7031.785,E2 -7031.785} C_VEL
LIN {X 0,Y 481.742,Z 57.476,A -85,B 0,C 180,E1 -7035.225,E2 -7035.225} C_VEL
LIN {X 0,Y 481.707,Z 57.477,A -85,B 0,C 180,E1 -7038.722,E2 -7038.722} C_VEL
LIN {X 0,Y 481.646,Z 57.493,A -85,B 0,C 180,E1 -7041.395,E2 -7041.395} C_VEL
LIN {X 0,Y 481.65,Z 57.484,A -85,B 0,C 180,E1 -7044.115,E2 -7044.115} C_VEL
LIN {X 0,Y 481.715,Z 57.483,A -85,B 0,C 180,E1 -7047.132,E2 -7047.132} C_VEL
LIN {X 0,Y 481.678,Z 57.482,A -85,B 0,C 180,E1 -7049.742,E2 -7049.742} C_VEL
LIN {X 0,Y 481.671,Z 57.485,A -85,B 0,C 180,E1 -7052.675,E2 -7052.675} C_VEL
LIN {X 0,Y 481.637,Z 57.486,A -85,B 0,C 180,E1 -7055.71,E2 -7055.71} C_VEL
LIN {X 0,Y 481.667,Z 57.49,A -85,B 0,C 180,E1 -7058.86,E2 -7058.86} C_VEL
LIN {X 0,Y 481.628,Z 57.488,A -85,B 0,C 180,E1 -7062.163,E2 -7062.163} C_VEL
LIN {X 0,Y 481.656,Z 57.483,A -85,B 0,C 180,E1 -7065.542,E2 -7065.542} C_VEL
LIN {X 0,Y 481.65,Z 57.487,A -85,B 0,C 180,E1 -7068.958,E2 -7068.958} C_VEL
LIN {X 0,Y 481.65,Z 57.487,A -85,B 0,C 180,E1 -7071.994,E2 -7071.994} C_VEL
LIN {X 0,Y 481.688,Z 57.479,A -85,B 0,C 180,E1 -7075.318,E2 -7075.318} C_VEL
LIN {X 0,Y 481.648,Z 57.492,A -85,B 0,C 180,E1 -7078.312,E2 -7078.312} C_VEL
LIN {X 0,Y 481.677,Z 57.481,A -85,B 0,C 180,E1 -7081.217,E2 -7081.217} C_VEL
LIN {X 0,Y 481.646,Z 57.489,A -85,B 0,C 180,E1 -7084.319,E2 -7084.319} C_VEL
LIN {X 0,Y 481.678,Z 57.481,A -85,B 0,C 180,E1 -7086.812,E2 -7086.812} C_VEL
LIN {X 0,Y 481.639,Z 57.488,A -85,B 0,C 180,E1 -7087.954,E2 -7087.954} C_VEL
LIN {X 0,Y 480.972,Z 57.571,A -85,B 0,C 180,E1 -7088.652,E2 -7088.652} C_VEL
LIN {X 0,Y 478.148,Z 57.927,A -85,B 0,C 180,E1 -7089.786,E2 -7089.786} C_VEL
LIN {X 0,Y 475.762,Z 58.221,A -85,B 0,C 180,E1 -7090.7,E2 -7090.7} C_VEL
LIN {X 0,Y 474.734,Z 58.348,A -85,B 0,C 180,E1 -7091.406,E2 -7091.406} C_VEL
LIN {X 0,Y 474.647,Z 58.361,A -85,B 0,C 180,E1 -7091.645,E2 -7091.645} C_VEL
LIN {X 0,Y 474.702,Z 58.354,A -85,B 0,C 180,E1 -7094.545,E2 -7094.545} C_VEL
LIN {X 0,Y 474.673,Z 58.406,A -85,B 0,C 180,E1 -7096.951,E2 -7096.951} C_VEL
LIN {X 0,Y 475.524,Z 64.394,A -85,B 0,C 180,E1 -7098.275,E2 -7098.275} C_VEL
LIN {X 0,Y 475.526,Z 74.647,A -85,B 0,C 180,E1 -7100.418,E2 -7100.418} C_VEL
LIN {X 0,Y 478.054,Z 88.275,A -85,B 0,C 180,E1 -7100.709,E2 -7100.709} C_VEL
LIN {X 0,Y 477.31,Z 181.061,A -85,B 0,C 180,E1 -7102.119,E2 -7102.119} C_VEL
LIN {X 0,Y 477.115,Z 194.193,A -85,B 0,C 180,E1 -7102.488,E2 -7102.488} C_VEL
LIN {X 0,Y 476.748,Z 206.824,A -85,B 0,C 180,E1 -7103.015,E2 -7103.015} C_VEL
LIN {X 0,Y 476.56,Z 218.018,A -85,B 0,C 180,E1 -7103.65,E2 -7103.65} C_VEL
LIN {X 0,Y 476.022,Z 229.608,A -85,B 0,C 180,E1 -7104.493,E2 -7104.493} C_VEL
LIN {X 0,Y 475.568,Z 240.005,A -85,B 0,C 180,E1 -7105.444,E2 -7105.444} C_VEL
LIN {X 0,Y 475.256,Z 248.504,A -85,B 0,C 180,E1 -7106.397,E2 -7106.397} C_VEL
LIN {X 0,Y 474.873,Z 256.358,A -85,B 0,C 180,E1 -7107.456,E2 -7107.456} C_VEL
LIN {X 0,Y 474.504,Z 264.066,A -85,B 0,C 180,E1 -7108.727,E2 -7108.727} C_VEL
LIN {X 0,Y 474.203,Z 270.238,A -85,B 0,C 180,E1 -7110,E2 -7110} C_VEL
LIN {X 0,Y 474.008,Z 275.153,A -85,B 0,C 180,E1 -7111.275,E2 -7111.275} C_VEL
LIN {X 0,Y 473.937,Z 278.957,A -85,B 0,C 180,E1 -7112.55,E2 -7112.55} C_VEL
LIN {X 0,Y 473.892,Z 280.922,A -85,B 0,C 180,E1 -7113.401,E2 -7113.401} C_VEL
LIN {X 0,Y 473.787,Z 282.483,A -85,B 0,C 180,E1 -7114.254,E2 -7114.254} C_VEL
LIN {X 0,Y 473.786,Z 283.619,A -85,B 0,C 180,E1 -7115.106,E2 -7115.106} C_VEL
LIN {X 0,Y 473.841,Z 284.574,A -85,B 0,C 180,E1 -7116.408,E2 -7116.408} C_VEL
LIN {X 0,Y 473.758,Z 284.612,A -85,B 0,C 180,E1 -7117.673,E2 -7117.673} C_VEL
LIN {X 0,Y 473.755,Z 284.155,A -85,B 0,C 180,E1 -7118.531,E2 -7118.531} C_VEL
LIN {X 0,Y 473.793,Z 281.987,A -85,B 0,C 180,E1 -7120.254,E2 -7120.254} C_VEL
LIN {X 0,Y 473.984,Z 278.449,A -85,B 0,C 180,E1 -7121.868,E2 -7121.868} C_VEL
LIN {X 0,Y 474.138,Z 273.976,A -85,B 0,C 180,E1 -7123.283,E2 -7123.283} C_VEL
LIN {X 0,Y 474.486,Z 267.599,A -85,B 0,C 180,E1 -7124.804,E2 -7124.804} C_VEL
LIN {X 0,Y 474.782,Z 260.373,A -85,B 0,C 180,E1 -7126.153,E2 -7126.153} C_VEL
LIN {X 0,Y 475.164,Z 251.764,A -85,B 0,C 180,E1 -7127.429,E2 -7127.429} C_VEL
LIN {X 0,Y 475.718,Z 241.667,A -85,B 0,C 180,E1 -7128.632,E2 -7128.632} C_VEL
LIN {X 0,Y 476.156,Z 231.269,A -85,B 0,C 180,E1 -7129.62,E2 -7129.62} C_VEL
LIN {X 0,Y 476.644,Z 219.655,A -85,B 0,C 180,E1 -7130.499,E2 -7130.499} C_VEL
LIN {X 0,Y 477.14,Z 207.448,A -85,B 0,C 180,E1 -7131.211,E2 -7131.211} C_VEL
LIN {X 0,Y 477.467,Z 194.452,A -85,B 0,C 180,E1 -7131.762,E2 -7131.762} C_VEL
LIN {X 0,Y 477.788,Z 181.424,A -85,B 0,C 180,E1 -7132.129,E2 -7132.129} C_VEL
LIN {X 0,Y 478.44,Z 87.539,A -85,B 0,C 180,E1 -7133.578,E2 -7133.578} C_VEL
LIN {X 0,Y 475.657,Z 74.605,A -85,B 0,C 180,E1 -7133.908,E2 -7133.908} C_VEL
LIN {X 0,Y 475.82,Z 65.086,A -85,B 0,C 180,E1 -7135.954,E2 -7135.954} C_VEL
LIN {X 0,Y 474.636,Z 58.364,A -85,B 0,C 180,E1 -7137.539,E2 -7137.539} C_VEL
LIN {X 0,Y 474.595,Z 58.368,A -85,B 0,C 180,E1 -7140.807,E2 -7140.807} C_VEL
LIN {X 0,Y 474.606,Z 58.371,A -85,B 0,C 180,E1 -7143.977,E2 -7143.977} C_VEL
LIN {X 0,Y 474.552,Z 58.37,A -85,B 0,C 180,E1 -7146.895,E2 -7146.895} C_VEL
LIN {X 0,Y 474.582,Z 58.371,A -85,B 0,C 180,E1 -7149.64,E2 -7149.64} C_VEL
LIN {X 0,Y 474.568,Z 58.368,A -85,B 0,C 180,E1 -7152.94,E2 -7152.94} C_VEL
LIN {X 0,Y 474.601,Z 58.366,A -85,B 0,C 180,E1 -7155.894,E2 -7155.894} C_VEL
LIN {X 0,Y 474.583,Z 58.365,A -85,B 0,C 180,E1 -7159.048,E2 -7159.048} C_VEL
LIN {X 0,Y 474.583,Z 58.37,A -85,B 0,C 180,E1 -7161.709,E2 -7161.709} C_VEL
LIN {X 0,Y 474.606,Z 58.361,A -85,B 0,C 180,E1 -7164.724,E2 -7164.724} C_VEL
LIN {X 0,Y 474.613,Z 58.361,A -85,B 0,C 180,E1 -7167.786,E2 -7167.786} C_VEL
LIN {X 0,Y 474.581,Z 58.369,A -85,B 0,C 180,E1 -7170.895,E2 -7170.895} C_VEL
LIN {X 0,Y 474.574,Z 58.368,A -85,B 0,C 180,E1 -7173.623,E2 -7173.623} C_VEL
LIN {X 0,Y 474.637,Z 58.361,A -85,B 0,C 180,E1 -7176.642,E2 -7176.642} C_VEL
LIN {X 0,Y 474.653,Z 58.357,A -85,B 0,C 180,E1 -7180.089,E2 -7180.089} C_VEL
LIN {X 0,Y 474.632,Z 58.36,A -85,B 0,C 180,E1 -7182.773,E2 -7182.773} C_VEL
LIN {X 0,Y 474.637,Z 58.359,A -85,B 0,C 180,E1 -7185.42,E2 -7185.42} C_VEL
LIN {X 0,Y 474.707,Z 58.346,A -85,B 0,C 180,E1 -7188.037,E2 -7188.037} C_VEL
LIN {X 0,Y 474.699,Z 58.35,A -85,B 0,C 180,E1 -7191.486,E2 -7191.486} C_VEL
LIN {X 0,Y 474.732,Z 58.345,A -85,B 0,C 180,E1 -7194.052,E2 -7194.052} C_VEL
LIN {X 0,Y 474.885,Z 58.328,A -85,B 0,C 180,E1 -7197.455,E2 -7197.455} C_VEL
LIN {X 0,Y 474.882,Z 58.327,A -85,B 0,C 180,E1 -7200,E2 -7200} C_VEL
LIN {X 0,Y 474.876,Z 58.331,A -85,B 0,C 180,E1 -7202.545,E2 -7202.545} C_VEL
LIN {X 0,Y 474.742,Z 58.345,A -85,B 0,C 180,E1 -7205.948,E2 -7205.948} C_VEL
LIN {X 0,Y 474.7,Z 58.351,A -85,B 0,C 180,E1 -7208.514,E2 -7208.514} C_VEL
LIN {X 0,Y 474.708,Z 58.35,A -85,B 0,C 180,E1 -7211.962,E2 -7211.962} C_VEL
LIN {X 0,Y 474.7,Z 58.356,A -85,B 0,C 180,E1 -7215.456,E2 -7215.456} C_VEL
LIN {X 0,Y 474.663,Z 58.355,A -85,B 0,C 180,E1 -7219.01,E2 -7219.01} C_VEL
LIN {X 0,Y 474.591,Z 58.363,A -85,B 0,C 180,E1 -7221.729,E2 -7221.729} C_VEL
LIN {X 0,Y 474.631,Z 58.359,A -85,B 0,C 180,E1 -7224.494,E2 -7224.494} C_VEL
LIN {X 0,Y 474.676,Z 58.357,A -85,B 0,C 180,E1 -7227.332,E2 -7227.332} C_VEL
LIN {X 0,Y 474.606,Z 58.361,A -85,B 0,C 180,E1 -7230.23,E2 -7230.23} C_VEL
LIN {X 0,Y 474.646,Z 58.362,A -85,B 0,C 180,E1 -7233.22,E2 -7233.22} C_VEL
LIN {X 0,Y 474.592,Z 58.357,A -85,B 0,C 180,E1 -7236.323,E2 -7236.323} C_VEL
LIN {X 0,Y 474.62,Z 58.361,A -85,B 0,C 180,E1 -7239.646,E2 -7239.646} C_VEL
LIN {X 0,Y 474.617,Z 58.366,A -85,B 0,C 180,E1 -7242.934,E2 -7242.934} C_VEL
LIN {X 0,Y 474.609,Z 58.362,A -85,B 0,C 180,E1 -7245.895,E2 -7245.895} C_VEL
LIN {X 0,Y 474.63,Z 58.36,A -85,B 0,C 180,E1 -7249.041,E2 -7249.041} C_VEL
LIN {X 0,Y 474.613,Z 58.362,A -85,B 0,C 180,E1 -7251.704,E2 -7251.704} C_VEL
LIN {X 0,Y 474.627,Z 58.362,A -85,B 0,C 180,E1 -7254.726,E2 -7254.726} C_VEL
LIN {X 0,Y 474.638,Z 58.366,A -85,B 0,C 180,E1 -7257.788,E2 -7257.788} C_VEL
LIN {X 0,Y 474.625,Z 58.364,A -85,B 0,C 180,E1 -7260.885,E2 -7260.885} C_VEL
LIN {X 0,Y 474.708,Z 58.502,A -85,B 0,C 180,E1 -7263.542,E2 -7263.542} C_VEL
LIN {X 0,Y 476.913,Z 69.669,A -85,B 0,C 180,E1 -7265.63,E2 -7265.63} C_VEL
LIN {X 0,Y 476.728,Z 78.976,A -85,B 0,C 180,E1 -7267.233,E2 -7267.233} C_VEL
LIN {X 0,Y 475.884,Z 97.722,A -85,B 0,C 180,E1 -7270.39,E2 -7270.39} C_VEL
LIN {X 0,Y 475.292,Z 114.15,A -85,B 0,C 180,E1 -7273.122,E2 -7273.122} C_VEL
LIN {X 0,Y 478.145,Z 133.344,A -85,B 0,C 180,E1 -7273.537,E2 -7273.537} C_VEL
LIN {X 0,Y 477.548,Z 222.636,A -85,B 0,C 180,E1 -7274.912,E2 -7274.912} C_VEL
LIN {X 0,Y 477.131,Z 235.929,A -85,B 0,C 180,E1 -7275.28,E2 -7275.28} C_VEL
LIN {X 0,Y 476.665,Z 248.668,A -85,B 0,C 180,E1 -7275.811,E2 -7275.811} C_VEL
LIN {X 0,Y 476.205,Z 260.004,A -85,B 0,C 180,E1 -7276.45,E2 -7276.45} C_VEL
LIN {X 0,Y 475.622,Z 272.058,A -85,B 0,C 180,E1 -7277.333,E2 -7277.333} C_VEL
LIN {X 0,Y 475.149,Z 283.28,A -85,B 0,C 180,E1 -7278.373,E2 -7278.373} C_VEL
LIN {X 0,Y 474.705,Z 291.71,A -85,B 0,C 180,E1 -7279.335,E2 -7279.335} C_VEL
LIN {X 0,Y 474.33,Z 300.868,A -85,B 0,C 180,E1 -7280.62,E2 -7280.62} C_VEL
LIN {X 0,Y 474.066,Z 308.26,A -85,B 0,C 180,E1 -7281.903,E2 -7281.903} C_VEL
LIN {X 0,Y 473.892,Z 314.201,A -85,B 0,C 180,E1 -7283.186,E2 -7283.186} C_VEL
LIN {X 0,Y 473.818,Z 318.898,A -85,B 0,C 180,E1 -7284.467,E2 -7284.467} C_VEL
LIN {X 0,Y 473.734,Z 322.484,A -85,B 0,C 180,E1 -7285.746,E2 -7285.746} C_VEL
LIN {X 0,Y 473.805,Z 324.331,A -85,B 0,C 180,E1 -7286.598,E2 -7286.598} C_VEL
LIN {X 0,Y 473.759,Z 326.703,A -85,B 0,C 180,E1 -7288.3,E2 -7288.3} C_VEL
LIN {X 0,Y 473.699,Z 327.301,A -85,B 0,C 180,E1 -7289.15,E2 -7289.15} C_VEL
LIN {X 0,Y 473.686,Z 327.497,A -85,B 0,C 180,E1 -7290,E2 -7290} C_VEL
LIN {X 0,Y 473.759,Z 326.646,A -85,B 0,C 180,E1 -7291.7,E2 -7291.7} C_VEL
LIN {X 0,Y 473.765,Z 325.634,A -85,B 0,C 180,E1 -7292.55,E2 -7292.55} C_VEL
LIN {X 0,Y 473.823,Z 324.211,A -85,B 0,C 180,E1 -7293.401,E2 -7293.401} C_VEL
LIN {X 0,Y 473.759,Z 321.231,A -85,B 0,C 180,E1 -7294.68,E2 -7294.68} C_VEL
LIN {X 0,Y 473.783,Z 317.2,A -85,B 0,C 180,E1 -7295.96,E2 -7295.96} C_VEL
LIN {X 0,Y 473.98,Z 310.997,A -85,B 0,C 180,E1 -7297.454,E2 -7297.454} C_VEL
LIN {X 0,Y 474.152,Z 304.225,A -85,B 0,C 180,E1 -7298.738,E2 -7298.738} C_VEL
LIN {X 0,Y 474.444,Z 295.822,A -85,B 0,C 180,E1 -7300.023,E2 -7300.023} C_VEL
LIN {X 0,Y 474.862,Z 287.17,A -85,B 0,C 180,E1 -7301.093,E2 -7301.093} C_VEL
LIN {X 0,Y 475.282,Z 276.941,A -85,B 0,C 180,E1 -7302.123,E2 -7302.123} C_VEL
LIN {X 0,Y 475.745,Z 265.903,A -85,B 0,C 180,E1 -7303.019,E2 -7303.019} C_VEL
LIN {X 0,Y 476.24,Z 254.163,A -85,B 0,C 180,E1 -7303.766,E2 -7303.766} C_VEL
LIN {X 0,Y 476.633,Z 241.942,A -85,B 0,C 180,E1 -7304.353,E2 -7304.353} C_VEL
LIN {X 0,Y 477.088,Z 229.545,A -85,B 0,C 180,E1 -7304.775,E2 -7304.775} C_VEL
LIN {X 0,Y 477.305,Z 217.22,A -85,B 0,C 180,E1 -7305.041,E2 -7305.041} C_VEL
LIN {X 0,Y 477.667,Z 132.144,A -85,B 0,C 180,E1 -7306.324,E2 -7306.324} C_VEL
LIN {X 0,Y 475.135,Z 114.267,A -85,B 0,C 180,E1 -7306.69,E2 -7306.69} C_VEL
LIN {X 0,Y 475.742,Z 96.262,A -85,B 0,C 180,E1 -7309.638,E2 -7309.638} C_VEL
LIN {X 0,Y 476.514,Z 75.904,A -85,B 0,C 180,E1 -7313.007,E2 -7313.007} C_VEL
LIN {X 0,Y 476.7,Z 69.423,A -85,B 0,C 180,E1 -7314.094,E2 -7314.094} C_VEL
LIN {X 0,Y 474.695,Z 58.359,A -85,B 0,C 180,E1 -7316.086,E2 -7316.086} C_VEL
LIN {X 0,Y 474.625,Z 58.362,A -85,B 0,C 180,E1 -7319.115,E2 -7319.115} C_VEL
LIN {X 0,Y 474.616,Z 58.362,A -85,B 0,C 180,E1 -7322.43,E2 -7322.43} C_VEL
LIN {X 0,Y 474.615,Z 58.364,A -85,B 0,C 180,E1 -7325.469,E2 -7325.469} C_VEL
LIN {X 0,Y 474.612,Z 58.361,A -85,B 0,C 180,E1 -7328.457,E2 -7328.457} C_VEL
LIN {X 0,Y 474.627,Z 58.36,A -85,B 0,C 180,E1 -7330.959,E2 -7330.959} C_VEL
LIN {X 0,Y 474.606,Z 58.363,A -85,B 0,C 180,E1 -7334.105,E2 -7334.105} C_VEL
LIN {X 0,Y 474.614,Z 58.364,A -85,B 0,C 180,E1 -7337.066,E2 -7337.066} C_VEL
LIN {X 0,Y 474.617,Z 58.36,A -85,B 0,C 180,E1 -7340.354,E2 -7340.354} C_VEL
LIN {X 0,Y 474.589,Z 58.366,A -85,B 0,C 180,E1 -7343.676,E2 -7343.676} C_VEL
LIN {X 0,Y 474.642,Z 58.36,A -85,B 0,C 180,E1 -7346.78,E2 -7346.78} C_VEL
LIN {X 0,Y 474.605,Z 58.362,A -85,B 0,C 180,E1 -7349.77,E2 -7349.77} C_VEL
LIN {X 0,Y 474.697,Z 58.355,A -85,B 0,C 180,E1 -7352.68,E2 -7352.68} C_VEL
LIN {X 0,Y 474.653,Z 58.357,A -85,B 0,C 180,E1 -7355.507,E2 -7355.507} C_VEL
LIN {X 0,Y 474.67,Z 58.356,A -85,B 0,C 180,E1 -7359.185,E2 -7359.185} C_VEL
LIN {X 0,Y 474.645,Z 58.357,A -85,B 0,C 180,E1 -7361.884,E2 -7361.884} C_VEL
LIN {X 0,Y 474.699,Z 58.358,A -85,B 0,C 180,E1 -7364.544,E2 -7364.544} C_VEL
LIN {X 0,Y 474.704,Z 58.352,A -85,B 0,C 180,E1 -7368.038,E2 -7368.038} C_VEL
LIN {X 0,Y 474.726,Z 58.347,A -85,B 0,C 180,E1 -7371.487,E2 -7371.487} C_VEL
LIN {X 0,Y 474.771,Z 58.346,A -85,B 0,C 180,E1 -7374.052,E2 -7374.052} C_VEL
LIN {X 0,Y 474.887,Z 58.327,A -85,B 0,C 180,E1 -7377.456,E2 -7377.456} C_VEL
LIN {X 0,Y 474.911,Z 58.33,A -85,B 0,C 180,E1 -7380,E2 -7380} C_VEL
LIN {X 0,Y 474.887,Z 58.328,A -85,B 0,C 180,E1 -7382.545,E2 -7382.545} C_VEL
LIN {X 0,Y 474.758,Z 58.35,A -85,B 0,C 180,E1 -7385.948,E2 -7385.948} C_VEL
LIN {X 0,Y 474.711,Z 58.349,A -85,B 0,C 180,E1 -7388.514,E2 -7388.514} C_VEL
LIN {X 0,Y 474.705,Z 58.354,A -85,B 0,C 180,E1 -7391.963,E2 -7391.963} C_VEL
LIN {X 0,Y 474.699,Z 58.356,A -85,B 0,C 180,E1 -7395.456,E2 -7395.456} C_VEL
LIN {X 0,Y 474.662,Z 58.357,A -85,B 0,C 180,E1 -7399.011,E2 -7399.011} C_VEL
LIN {X 0,Y 474.588,Z 58.368,A -85,B 0,C 180,E1 -7401.729,E2 -7401.729} C_VEL
LIN {X 0,Y 474.629,Z 58.359,A -85,B 0,C 180,E1 -7404.495,E2 -7404.495} C_VEL
LIN {X 0,Y 474.674,Z 58.36,A -85,B 0,C 180,E1 -7407.333,E2 -7407.333} C_VEL
LIN {X 0,Y 474.604,Z 58.362,A -85,B 0,C 180,E1 -7410.231,E2 -7410.231} C_VEL
LIN {X 0,Y 474.626,Z 58.365,A -85,B 0,C 180,E1 -7413.222,E2 -7413.222} C_VEL
LIN {X 0,Y 474.59,Z 58.365,A -85,B 0,C 180,E1 -7416.324,E2 -7416.324} C_VEL
LIN {X 0,Y 474.622,Z 58.36,A -85,B 0,C 180,E1 -7419.549,E2 -7419.549} C_VEL
LIN {X 0,Y 474.587,Z 58.366,A -85,B 0,C 180,E1 -7422.232,E2 -7422.232} C_VEL
LIN {X 0,Y 474.618,Z 58.361,A -85,B 0,C 180,E1 -7425.298,E2 -7425.298} C_VEL
LIN {X 0,Y 474.616,Z 58.364,A -85,B 0,C 180,E1 -7428.214,E2 -7428.214} C_VEL
LIN {X 0,Y 474.611,Z 58.361,A -85,B 0,C 180,E1 -7431.543,E2 -7431.543} C_VEL
LIN {X 0,Y 474.622,Z 58.363,A -85,B 0,C 180,E1 -7434.726,E2 -7434.726} C_VEL
LIN {X 0,Y 474.638,Z 58.36,A -85,B 0,C 180,E1 -7437.788,E2 -7437.788} C_VEL
LIN {X 0,Y 474.61,Z 58.362,A -85,B 0,C 180,E1 -7440.889,E2 -7440.889} C_VEL
LIN {X 0,Y 474.593,Z 58.366,A -85,B 0,C 180,E1 -7443.625,E2 -7443.625} C_VEL
LIN {X 0,Y 474.638,Z 58.359,A -85,B 0,C 180,E1 -7446.642,E2 -7446.642} C_VEL
LIN {X 0,Y 474.655,Z 58.361,A -85,B 0,C 180,E1 -7450.09,E2 -7450.09} C_VEL
LIN {X 0,Y 474.647,Z 58.361,A -85,B 0,C 180,E1 -7451.645,E2 -7451.645} C_VEL
LIN {X 0,Y 473.976,Z 58.451,A -85,B 0,C 180,E1 -7452.354,E2 -7452.354} C_VEL
LIN {X 0,Y 471.129,Z 58.808,A -85,B 0,C 180,E1 -7453.506,E2 -7453.506} C_VEL
